    |   movel([0.102355, -1.292766, -2.631086, -0.788537, 1.570796, 1.673152],accel_mss,speed_ms,0,blend_radius_m)
    |   movel([0.101965, -1.293057, -2.630916, -0.788416, 1.570796, 1.672761],accel_mss,speed_ms,0,blend_radius_m)
    |   movel([0.101499, -1.293216, -2.630823, -0.788350, 1.570796, 1.672295],accel_mss,speed_ms,0,blend_radius_m)
    |   movel([0.101150, -1.293383, -2.630725, -0.788281, 1.570796, 1.671947],accel_mss,speed_ms,0,blend_radius_m)
    |   movel([0.100675, -1.293364, -2.630736, -0.788289, 1.570796, 1.671471],accel_mss,speed_ms,0,blend_radius_m)
    |   movel([0.100391, -1.293407, -2.630711, -0.788271, 1.570796, 1.671188],accel_mss,speed_ms,0,blend_radius_m)
    |   movel([0.100053, -1.293699, -2.630540, -0.788150, 1.570796, 1.670849],accel_mss,speed_ms,0,blend_radius_m)
    |   movel([0.100321, -1.293715, -2.630530, -0.788144, 1.570796, 1.671118],accel_mss,speed_ms,0,blend_radius_m)
    |   movel([0.100651, -1.293667, -2.630559, -0.788164, 1.570796, 1.671448],accel_mss,speed_ms,0,blend_radius_m)
    |   movel([0.101031, -1.293650, -2.630569, -0.788171, 1.570796, 1.671827],accel_mss,speed_ms,0,blend_radius_m)
    |   movel([0.101319, -1.293615, -2.630589, -0.788185, 1.570796, 1.672116],accel_mss,speed_ms,0,blend_radius_m)
    |   movel([0.101619, -1.293570, -2.630615, -0.788204, 1.570796, 1.672416],accel_mss,speed_ms,0,blend_radius_m)
    |   movel([0.102043, -1.293494, -2.630660, -0.788235, 1.570796, 1.672840],accel_mss,speed_ms,0,blend_radius_m)
    |   movel([0.101987, -1.293260, -2.630797, -0.788332, 1.570796, 1.672784],accel_mss,speed_ms,0,blend_radius_m)
    |   movel([0.102373, -1.293289, -2.630780, -0.788320, 1.570796, 1.673169],accel_mss,speed_ms,0,blend_radius_m)
    |   movel([0.102475, -1.293491, -2.630662, -0.788236, 1.570796, 1.673271],accel_mss,speed_ms,0,blend_radius_m)
    |   movel([0.102816, -1.293437, -2.630693, -0.788259, 1.570796, 1.673613],accel_mss,speed_ms,0,blend_radius_m)
    |   movel([0.103104, -1.293401, -2.630715, -0.788274, 1.570796, 1.673901],accel_mss,speed_ms,0,blend_radius_m)
    |   movel([0.103382, -1.293344, -2.630748, -0.788297, 1.570796, 1.674178],accel_mss,speed_ms,0,blend_radius_m)
    |   movel([0.103678, -1.293105, -2.630888, -0.788396, 1.570796, 1.674474],accel_mss,speed_ms,0,blend_radius_m)
    |   movel([0.103359, -1.293263, -2.630795, -0.788331, 1.570796, 1.674155],accel_mss,speed_ms,0,blend_radius_m)
    |   movel([0.103194, -1.293136, -2.630870, -0.788383, 1.570796, 1.673991],accel_mss,speed_ms,0,blend_radius_m)
    |   movel([0.103230, -1.292829, -2.631049, -0.788511, 1.570796, 1.674026],accel_mss,speed_ms,0,blend_radius_m)
    |   movel([0.103561, -1.292519, -2.631231, -0.788639, 1.570796, 1.674358],accel_mss,speed_ms,0,blend_radius_m)
    |   movel([0.103869, -1.292455, -2.631268, -0.788666, 1.570796, 1.674665],accel_mss,speed_ms,0,blend_radius_m)
    |   movel([0.103902, -1.292696, -2.631127, -0.788566, 1.570796, 1.674699],accel_mss,speed_ms,0,blend_radius_m)
    |   movel([0.104086, -1.292889, -2.631014, -0.788486, 1.570796, 1.674882],accel_mss,speed_ms,0,blend_radius_m)
    |   movel([0.104470, -1.293089, -2.630897, -0.788403, 1.570796, 1.675266],accel_mss,speed_ms,0,blend_radius_m)
    |   movel([0.104480, -1.293409, -2.630709, -0.788270, 1.570796, 1.675276],accel_mss,speed_ms,0,blend_radius_m)
    |   movel([0.104166, -1.293506, -2.630653, -0.788230, 1.570796, 1.674962],accel_mss,speed_ms,0,blend_radius_m)
    |   movel([0.103943, -1.293445, -2.630688, -0.788255, 1.570796, 1.674739],accel_mss,speed_ms,0,blend_radius_m)
    |   movel([0.103724, -1.293307, -2.630769, -0.788313, 1.570796, 1.674520],accel_mss,speed_ms,0,blend_radius_m)
    |   movel([0.103804, -1.293583, -2.630608, -0.788198, 1.570796, 1.674600],accel_mss,speed_ms,0,blend_radius_m)
    |   movel([0.103792, -1.293977, -2.630377, -0.788035, 1.570796, 1.674589],accel_mss,speed_ms,0,blend_radius_m)
    |   movel([0.103523, -1.294338, -2.630165, -0.787886, 1.570796, 1.674319],accel_mss,speed_ms,0,blend_radius_m)
    |   movel([0.103297, -1.294618, -2.630001, -0.787771, 1.570796, 1.674094],accel_mss,speed_ms,0,blend_radius_m)
    |   movel([0.102982, -1.294687, -2.629960, -0.787742, 1.570796, 1.673778],accel_mss,speed_ms,0,blend_radius_m)
    |   movel([0.102668, -1.294988, -2.629783, -0.787618, 1.570796, 1.673465],accel_mss,speed_ms,0,blend_radius_m)
    |   movel([0.102281, -1.295194, -2.629662, -0.787533, 1.570796, 1.673077],accel_mss,speed_ms,0,blend_radius_m)
    |   movel([0.101902, -1.295350, -2.629570, -0.787469, 1.570796, 1.672698],accel_mss,speed_ms,0,blend_radius_m)
    |   movel([0.101557, -1.295489, -2.629488, -0.787412, 1.570796, 1.672353],accel_mss,speed_ms,0,blend_radius_m)
    |   movel([0.101243, -1.295617, -2.629413, -0.787359, 1.570796, 1.672039],accel_mss,speed_ms,0,blend_radius_m)
    |   movel([0.101286, -1.295842, -2.629280, -0.787267, 1.570796, 1.672083],accel_mss,speed_ms,0,blend_radius_m)
    |   movel([0.100997, -1.295991, -2.629193, -0.787206, 1.570796, 1.671793],accel_mss,speed_ms,0,blend_radius_m)
    |   movel([0.100718, -1.295951, -2.629216, -0.787222, 1.570796, 1.671514],accel_mss,speed_ms,0,blend_radius_m)
    |   movel([0.100425, -1.296077, -2.629142, -0.787170, 1.570796, 1.671222],accel_mss,speed_ms,0,blend_radius_m)
    |   movel([0.099331, -1.296580, -2.628845, -0.786964, 1.570796, 1.670127],accel_mss,speed_ms,0,blend_radius_m)
    |   movel([0.097242, -1.297292, -2.628425, -0.786672, 1.570796, 1.668038],accel_mss,speed_ms,0,blend_radius_m)
    |   movel([0.095038, -1.297963, -2.628028, -0.786398, 1.570796, 1.665834],accel_mss,speed_ms,0,blend_radius_m)
    |   movel([0.093267, -1.298398, -2.627770, -0.786220, 1.570796, 1.664064],accel_mss,speed_ms,0,blend_radius_m)
    |   movel([0.092796, -1.298507, -2.627706, -0.786176, 1.570796, 1.663592],accel_mss,speed_ms,0,blend_radius_m)
    |   movel([0.092505, -1.298577, -2.627664, -0.786148, 1.570796, 1.663301],accel_mss,speed_ms,0,blend_radius_m)
    |   movel([0.092006, -1.298695, -2.627594, -0.786099, 1.570796, 1.662802],accel_mss,speed_ms,0,blend_radius_m)
    |   movel([0.091686, -1.298709, -2.627586, -0.786094, 1.570796, 1.662483],accel_mss,speed_ms,0,blend_radius_m)
    |   movel([0.091516, -1.298549, -2.627681, -0.786159, 1.570796, 1.662312],accel_mss,speed_ms,0,blend_radius_m)
    |   movel([0.090908, -1.298604, -2.627648, -0.786137, 1.570796, 1.661704],accel_mss,speed_ms,0,blend_radius_m)
    |   movel([0.091012, -1.298791, -2.627537, -0.786060, 1.570796, 1.661808],accel_mss,speed_ms,0,blend_radius_m)
    |   movel([0.091131, -1.298957, -2.627439, -0.785993, 1.570796, 1.661927],accel_mss,speed_ms,0,blend_radius_m)
    |   movel([0.091380, -1.299030, -2.627396, -0.785963, 1.570796, 1.662176],accel_mss,speed_ms,0,blend_radius_m)
    |   movel([0.091703, -1.299034, -2.627394, -0.785962, 1.570796, 1.662500],accel_mss,speed_ms,0,blend_radius_m)
    |   movel([0.091970, -1.298785, -2.627541, -0.786063, 1.570796, 1.662766],accel_mss,speed_ms,0,blend_radius_m)
    |   movel([0.092331, -1.298807, -2.627528, -0.786054, 1.570796, 1.663127],accel_mss,speed_ms,0,blend_radius_m)
    |   movel([0.092659, -1.298717, -2.627581, -0.786090, 1.570796, 1.663455],accel_mss,speed_ms,0,blend_radius_m)
    |   movel([0.092762, -1.298900, -2.627473, -0.786016, 1.570796, 1.663559],accel_mss,speed_ms,0,blend_radius_m)
    |   movel([0.092991, -1.298961, -2.627436, -0.785991, 1.570796, 1.663787],accel_mss,speed_ms,0,blend_radius_m)
    |   movel([0.093296, -1.298783, -2.627542, -0.786064, 1.570796, 1.664092],accel_mss,speed_ms,0,blend_radius_m)
    |   movel([0.093554, -1.298769, -2.627551, -0.786070, 1.570796, 1.664350],accel_mss,speed_ms,0,blend_radius_m)
    |   movel([0.093259, -1.299029, -2.627397, -0.785964, 1.570796, 1.664056],accel_mss,speed_ms,0,blend_radius_m)
    |   movel([0.092956, -1.299112, -2.627347, -0.785930, 1.570796, 1.663753],accel_mss,speed_ms,0,blend_radius_m)
    |   movel([0.092691, -1.299070, -2.627372, -0.785947, 1.570796, 1.663487],accel_mss,speed_ms,0,blend_radius_m)
    |   movel([0.092356, -1.298978, -2.627427, -0.785984, 1.570796, 1.663152],accel_mss,speed_ms,0,blend_radius_m)
    |   movel([0.092063, -1.299023, -2.627400, -0.785966, 1.570796, 1.662859],accel_mss,speed_ms,0,blend_radius_m)
    |   movel([0.091652, -1.299143, -2.627329, -0.785917, 1.570796, 1.662448],accel_mss,speed_ms,0,blend_radius_m)
    |   movel([0.091327, -1.299231, -2.627276, -0.785881, 1.570796, 1.662123],accel_mss,speed_ms,0,blend_radius_m)
    |   movel([0.091035, -1.299288, -2.627243, -0.785858, 1.570796, 1.661832],accel_mss,speed_ms,0,blend_radius_m)
    |   movel([0.090721, -1.299331, -2.627217, -0.785841, 1.570796, 1.661517],accel_mss,speed_ms,0,blend_radius_m)
    |   movel([0.090684, -1.299094, -2.627358, -0.785937, 1.570796, 1.661480],accel_mss,speed_ms,0,blend_radius_m)
    |   movel([0.090510, -1.298965, -2.627434, -0.785990, 1.570796, 1.661306],accel_mss,speed_ms,0,blend_radius_m)
    |   movel([0.090188, -1.299079, -2.627367, -0.785943, 1.570796, 1.660984],accel_mss,speed_ms,0,blend_radius_m)
    |   movel([0.090012, -1.298940, -2.627449, -0.786000, 1.570796, 1.660808],accel_mss,speed_ms,0,blend_radius_m)
    |   movel([0.089943, -1.298729, -2.627574, -0.786086, 1.570796, 1.660739],accel_mss,speed_ms,0,blend_radius_m)
    |   movel([0.089712, -1.298679, -2.627604, -0.786106, 1.570796, 1.660509],accel_mss,speed_ms,0,blend_radius_m)
    |   movel([0.089970, -1.298437, -2.627747, -0.786205, 1.570796, 1.660766],accel_mss,speed_ms,0,blend_radius_m)
    |   movel([0.090285, -1.298394, -2.627773, -0.786222, 1.570796, 1.661081],accel_mss,speed_ms,0,blend_radius_m)
    |   movel([0.090132, -1.298683, -2.627602, -0.786105, 1.570796, 1.660928],accel_mss,speed_ms,0,blend_radius_m)
    |   movel([0.090205, -1.298963, -2.627436, -0.785991, 1.570796, 1.661001],accel_mss,speed_ms,0,blend_radius_m)
    |   movel([0.090261, -1.298678, -2.627605, -0.786107, 1.570796, 1.661057],accel_mss,speed_ms,0,blend_radius_m)
    |   movel([0.090563, -1.298554, -2.627678, -0.786157, 1.570796, 1.661359],accel_mss,speed_ms,0,blend_radius_m)
    |   movel([0.090470, -1.298342, -2.627804, -0.786244, 1.570796, 1.661266],accel_mss,speed_ms,0,blend_radius_m)
    |   movel([0.090383, -1.298068, -2.627966, -0.786355, 1.570796, 1.661179],accel_mss,speed_ms,0,blend_radius_m)
    |   movel([0.090678, -1.297826, -2.628109, -0.786454, 1.570796, 1.661474],accel_mss,speed_ms,0,blend_radius_m)
    |   movel([0.090825, -1.297494, -2.628306, -0.786590, 1.570796, 1.661621],accel_mss,speed_ms,0,blend_radius_m)
    |   movel([0.090518, -1.297690, -2.628189, -0.786509, 1.570796, 1.661314],accel_mss,speed_ms,0,blend_radius_m)
    |   movel([0.090290, -1.297927, -2.628049, -0.786413, 1.570796, 1.661086],accel_mss,speed_ms,0,blend_radius_m)
    |   movel([0.090113, -1.298212, -2.627880, -0.786296, 1.570796, 1.660910],accel_mss,speed_ms,0,blend_radius_m)
    |   movel([0.089804, -1.298280, -2.627840, -0.786269, 1.570796, 1.660600],accel_mss,speed_ms,0,blend_radius_m)
    |   movel([0.089954, -1.297963, -2.628028, -0.786398, 1.570796, 1.660750],accel_mss,speed_ms,0,blend_radius_m)
    |   movel([0.090167, -1.297691, -2.628189, -0.786509, 1.570796, 1.660963],accel_mss,speed_ms,0,blend_radius_m)
    |   movel([0.090457, -1.297347, -2.628392, -0.786650, 1.570796, 1.661253],accel_mss,speed_ms,0,blend_radius_m)
    |   movel([0.090350, -1.297056, -2.628564, -0.786769, 1.570796, 1.661146],accel_mss,speed_ms,0,blend_radius_m)
    |   movel([0.090002, -1.296971, -2.628614, -0.786803, 1.570796, 1.660798],accel_mss,speed_ms,0,blend_radius_m)
    |   movel([0.089628, -1.296935, -2.628635, -0.786818, 1.570796, 1.660424],accel_mss,speed_ms,0,blend_radius_m)
    |   movel([0.089304, -1.296977, -2.628611, -0.786801, 1.570796, 1.660101],accel_mss,speed_ms,0,blend_radius_m)
    |   movel([0.089032, -1.296934, -2.628637, -0.786819, 1.570796, 1.659829],accel_mss,speed_ms,0,blend_radius_m)
    |   movel([0.088749, -1.296974, -2.628613, -0.786802, 1.570796, 1.659546],accel_mss,speed_ms,0,blend_radius_m)
    |   movel([0.088519, -1.296916, -2.628647, -0.786826, 1.570796, 1.659315],accel_mss,speed_ms,0,blend_radius_m)
    |   movel([0.088260, -1.296793, -2.628720, -0.786877, 1.570796, 1.659057],accel_mss,speed_ms,0,blend_radius_m)
    |   movel([0.087984, -1.296604, -2.628831, -0.786954, 1.570796, 1.658780],accel_mss,speed_ms,0,blend_radius_m)
    |   movel([0.087838, -1.296402, -2.628950, -0.787037, 1.570796, 1.658634],accel_mss,speed_ms,0,blend_radius_m)
    |   movel([0.087930, -1.296130, -2.629111, -0.787148, 1.570796, 1.658726],accel_mss,speed_ms,0,blend_radius_m)
    |   movel([0.088018, -1.295835, -2.629284, -0.787270, 1.570796, 1.658814],accel_mss,speed_ms,0,blend_radius_m)
    |   movel([0.088177, -1.295298, -2.629600, -0.787490, 1.570796, 1.658973],accel_mss,speed_ms,0,blend_radius_m)
    |   movel([0.088520, -1.294882, -2.629845, -0.787662, 1.570796, 1.659316],accel_mss,speed_ms,0,blend_radius_m)
    |   movel([0.088850, -1.294590, -2.630017, -0.787782, 1.570796, 1.659647],accel_mss,speed_ms,0,blend_radius_m)
    |   movel([0.089096, -1.294365, -2.630149, -0.787875, 1.570796, 1.659893],accel_mss,speed_ms,0,blend_radius_m)
    |   movel([0.089150, -1.293993, -2.630367, -0.788029, 1.570796, 1.659946],accel_mss,speed_ms,0,blend_radius_m)
    |   movel([0.088850, -1.293957, -2.630389, -0.788044, 1.570796, 1.659646],accel_mss,speed_ms,0,blend_radius_m)
    |   movel([0.088651, -1.293819, -2.630469, -0.788100, 1.570796, 1.659447],accel_mss,speed_ms,0,blend_radius_m)
    |   movel([0.088309, -1.293899, -2.630422, -0.788068, 1.570796, 1.659105],accel_mss,speed_ms,0,blend_radius_m)
    |   movel([0.087687, -1.293983, -2.630373, -0.788033, 1.570796, 1.658483],accel_mss,speed_ms,0,blend_radius_m)
    |   movel([0.087026, -1.293852, -2.630450, -0.788087, 1.570796, 1.657823],accel_mss,speed_ms,0,blend_radius_m)
    |   movel([0.086481, -1.293564, -2.630619, -0.788206, 1.570796, 1.657277],accel_mss,speed_ms,0,blend_radius_m)
    |   movel([0.086205, -1.293166, -2.630852, -0.788371, 1.570796, 1.657001],accel_mss,speed_ms,0,blend_radius_m)
    |   movel([0.086167, -1.292865, -2.631028, -0.788496, 1.570796, 1.656963],accel_mss,speed_ms,0,blend_radius_m)
    |   movel([0.086235, -1.292549, -2.631213, -0.788627, 1.570796, 1.657032],accel_mss,speed_ms,0,blend_radius_m)
    |   movel([0.086426, -1.292178, -2.631430, -0.788781, 1.570796, 1.657222],accel_mss,speed_ms,0,blend_radius_m)
    |   movel([0.086757, -1.291717, -2.631699, -0.788973, 1.570796, 1.657553],accel_mss,speed_ms,0,blend_radius_m)
    |   movel([0.086981, -1.291477, -2.631839, -0.789073, 1.570796, 1.657777],accel_mss,speed_ms,0,blend_radius_m)
    |   movel([0.087305, -1.291207, -2.631997, -0.789185, 1.570796, 1.658101],accel_mss,speed_ms,0,blend_radius_m)
    |   movel([0.087627, -1.290981, -2.632129, -0.789279, 1.570796, 1.658423],accel_mss,speed_ms,0,blend_radius_m)
    |   movel([0.087930, -1.290792, -2.632238, -0.789358, 1.570796, 1.658726],accel_mss,speed_ms,0,blend_radius_m)
    |   movel([0.088216, -1.290788, -2.632241, -0.789360, 1.570796, 1.659013],accel_mss,speed_ms,0,blend_radius_m)
    |   movel([0.088406, -1.290922, -2.632163, -0.789304, 1.570796, 1.659202],accel_mss,speed_ms,0,blend_radius_m)
    |   movel([0.088248, -1.290579, -2.632363, -0.789447, 1.570796, 1.659044],accel_mss,speed_ms,0,blend_radius_m)
    |   movel([0.088513, -1.290389, -2.632473, -0.789526, 1.570796, 1.659309],accel_mss,speed_ms,0,blend_radius_m)
    |   movel([0.088853, -1.290071, -2.632658, -0.789660, 1.570796, 1.659650],accel_mss,speed_ms,0,blend_radius_m)
    |   movel([0.089467, -1.289643, -2.632907, -0.789839, 1.570796, 1.660263],accel_mss,speed_ms,0,blend_radius_m)
    |   movel([0.090092, -1.289248, -2.633137, -0.790004, 1.570796, 1.660888],accel_mss,speed_ms,0,blend_radius_m)
    |   movel([0.090426, -1.289175, -2.633179, -0.790035, 1.570796, 1.661223],accel_mss,speed_ms,0,blend_radius_m)
    |   movel([0.090517, -1.289419, -2.633037, -0.789932, 1.570796, 1.661314],accel_mss,speed_ms,0,blend_radius_m)
    |   speed_ms = 0.003
    |   movel([0.090517, -1.275491, -2.626410, -0.810488, 1.570796, 1.661314],accel_mss,speed_ms,0,blend_radius_m)
    |   speed_ms = 1.000
    |   movel([0.090517, -1.248993, -2.612771, -0.850625, 1.570796, 1.661314],accel_mss,speed_ms,0,blend_radius_m)
    |   movel([0.108394, -1.243984, -2.615506, -0.852900, 1.570796, 1.679191],accel_mss,speed_ms,0,blend_radius_m)
    |   movel([0.108394, -1.270545, -2.629211, -0.812633, 1.570796, 1.679191],accel_mss,speed_ms,0,blend_radius_m)
    |   speed_ms = 0.003
    |   movel([0.108394, -1.280978, -2.634218, -0.797193, 1.570796, 1.679191],accel_mss,speed_ms,0,blend_radius_m)
    |   speed_ms = 0.007
    |   movel([0.108672, -1.280919, -2.634252, -0.797218, 1.570796, 1.679468],accel_mss,speed_ms,0,blend_radius_m)
    |   movel([0.108972, -1.280870, -2.634280, -0.797239, 1.570796, 1.679768],accel_mss,speed_ms,0,blend_radius_m)
    |   movel([0.108590, -1.281076, -2.634162, -0.797151, 1.570796, 1.679387],accel_mss,speed_ms,0,blend_radius_m)
    |   movel([0.108394, -1.280978, -2.634218, -0.797193, 1.570796, 1.679191],accel_mss,speed_ms,0,blend_radius_m)
    |   speed_ms = 0.003
    |   movel([0.108394, -1.284514, -2.635871, -0.792004, 1.570796, 1.679191],accel_mss,speed_ms,0,blend_radius_m)
    |   speed_ms = 0.007
    |   movel([0.108672, -1.284455, -2.635905, -0.792029, 1.570796, 1.679468],accel_mss,speed_ms,0,blend_radius_m)
    |   movel([0.108972, -1.284406, -2.635933, -0.792050, 1.570796, 1.679768],accel_mss,speed_ms,0,blend_radius_m)
    |   movel([0.108590, -1.284612, -2.635815, -0.791962, 1.570796, 1.679387],accel_mss,speed_ms,0,blend_radius_m)
    |   movel([0.108394, -1.284514, -2.635871, -0.792004, 1.570796, 1.679191],accel_mss,speed_ms,0,blend_radius_m)
    |   speed_ms = 0.003
    |   movel([0.108394, -1.270545, -2.629211, -0.812633, 1.570796, 1.679191],accel_mss,speed_ms,0,blend_radius_m)
    |   speed_ms = 1.000
    |   movel([0.108394, -1.243984, -2.615506, -0.852900, 1.570796, 1.679191],accel_mss,speed_ms,0,blend_radius_m)
    |   movel([0.134199, -1.228063, -2.624004, -0.860322, 1.570796, 1.704996],accel_mss,speed_ms,0,blend_radius_m)
    |   movel([0.134199, -1.254817, -2.637919, -0.819653, 1.570796, 1.704996],accel_mss,speed_ms,0,blend_radius_m)
    |   speed_ms = 0.003
    |   movel([0.134199, -1.265339, -2.643007, -0.804044, 1.570796, 1.704996],accel_mss,speed_ms,0,blend_radius_m)
    |   speed_ms = 0.007
    |   movel([0.134398, -1.265029, -2.643178, -0.804183, 1.570796, 1.705194],accel_mss,speed_ms,0,blend_radius_m)
    |   movel([0.134745, -1.264784, -2.643313, -0.804292, 1.570796, 1.705541],accel_mss,speed_ms,0,blend_radius_m)
    |   movel([0.135237, -1.264642, -2.643391, -0.804356, 1.570796, 1.706033],accel_mss,speed_ms,0,blend_radius_m)
    |   movel([0.135651, -1.264639, -2.643393, -0.804357, 1.570796, 1.706448],accel_mss,speed_ms,0,blend_radius_m)
    |   movel([0.135748, -1.264848, -2.643278, -0.804264, 1.570796, 1.706545],accel_mss,speed_ms,0,blend_radius_m)
    |   movel([0.135483, -1.265183, -2.643092, -0.804113, 1.570796, 1.706279],accel_mss,speed_ms,0,blend_radius_m)
    |   movel([0.135213, -1.265424, -2.642960, -0.804005, 1.570796, 1.706009],accel_mss,speed_ms,0,blend_radius_m)
    |   movel([0.134898, -1.265584, -2.642871, -0.803934, 1.570796, 1.705694],accel_mss,speed_ms,0,blend_radius_m)
    |   movel([0.134599, -1.265633, -2.642844, -0.803912, 1.570796, 1.705396],accel_mss,speed_ms,0,blend_radius_m)
    |   movel([0.134371, -1.265561, -2.642884, -0.803944, 1.570796, 1.705167],accel_mss,speed_ms,0,blend_radius_m)
    |   movel([0.134199, -1.265339, -2.643007, -0.804044, 1.570796, 1.704996],accel_mss,speed_ms,0,blend_radius_m)
    |   speed_ms = 0.003
    |   movel([0.134199, -1.268907, -2.644686, -0.798796, 1.570796, 1.704996],accel_mss,speed_ms,0,blend_radius_m)
    |   speed_ms = 0.007
    |   movel([0.134398, -1.268597, -2.644858, -0.798934, 1.570796, 1.705194],accel_mss,speed_ms,0,blend_radius_m)
    |   movel([0.134745, -1.268352, -2.644993, -0.799043, 1.570796, 1.705541],accel_mss,speed_ms,0,blend_radius_m)
    |   movel([0.135237, -1.268211, -2.645072, -0.799106, 1.570796, 1.706033],accel_mss,speed_ms,0,blend_radius_m)
    |   movel([0.135651, -1.268209, -2.645073, -0.799107, 1.570796, 1.706448],accel_mss,speed_ms,0,blend_radius_m)
    |   movel([0.135748, -1.268416, -2.644958, -0.799015, 1.570796, 1.706545],accel_mss,speed_ms,0,blend_radius_m)
    |   movel([0.135483, -1.268752, -2.644772, -0.798865, 1.570796, 1.706279],accel_mss,speed_ms,0,blend_radius_m)
    |   movel([0.135213, -1.268992, -2.644639, -0.798758, 1.570796, 1.706009],accel_mss,speed_ms,0,blend_radius_m)
    |   movel([0.134898, -1.269152, -2.644550, -0.798687, 1.570796, 1.705694],accel_mss,speed_ms,0,blend_radius_m)
    |   movel([0.134599, -1.269200, -2.644523, -0.798666, 1.570796, 1.705396],accel_mss,speed_ms,0,blend_radius_m)
    |   movel([0.134371, -1.269128, -2.644563, -0.798698, 1.570796, 1.705167],accel_mss,speed_ms,0,blend_radius_m)
    |   movel([0.134199, -1.268907, -2.644686, -0.798796, 1.570796, 1.704996],accel_mss,speed_ms,0,blend_radius_m)
    |   speed_ms = 0.003
    |   movel([0.134199, -1.254817, -2.637919, -0.819653, 1.570796, 1.704996],accel_mss,speed_ms,0,blend_radius_m)
    |   speed_ms = 1.000
    |   movel([0.134199, -1.228063, -2.624004, -0.860322, 1.570796, 1.704996],accel_mss,speed_ms,0,blend_radius_m)
    |   movel([0.135018, -1.226764, -2.624685, -0.860940, 1.570796, 1.705815],accel_mss,speed_ms,0,blend_radius_m)
    |   movel([0.135018, -1.253533, -2.638617, -0.820240, 1.570796, 1.705815],accel_mss,speed_ms,0,blend_radius_m)
    |   speed_ms = 0.003
    |   movel([0.135018, -1.264062, -2.643711, -0.804616, 1.570796, 1.705815],accel_mss,speed_ms,0,blend_radius_m)
    |   speed_ms = 0.007
    |   movel([0.133569, -1.264514, -2.643462, -0.804413, 1.570796, 1.704366],accel_mss,speed_ms,0,blend_radius_m)
    |   movel([0.132754, -1.264606, -2.643411, -0.804372, 1.570796, 1.703551],accel_mss,speed_ms,0,blend_radius_m)
    |   movel([0.132393, -1.264541, -2.643447, -0.804401, 1.570796, 1.703189],accel_mss,speed_ms,0,blend_radius_m)
    |   movel([0.132220, -1.264399, -2.643525, -0.804465, 1.570796, 1.703016],accel_mss,speed_ms,0,blend_radius_m)
    |   movel([0.132406, -1.263908, -2.643795, -0.804685, 1.570796, 1.703203],accel_mss,speed_ms,0,blend_radius_m)
    |   movel([0.132616, -1.263631, -2.643948, -0.804810, 1.570796, 1.703412],accel_mss,speed_ms,0,blend_radius_m)
    |   movel([0.132602, -1.263320, -2.644119, -0.804950, 1.570796, 1.703398],accel_mss,speed_ms,0,blend_radius_m)
    |   movel([0.132363, -1.263216, -2.644176, -0.804997, 1.570796, 1.703159],accel_mss,speed_ms,0,blend_radius_m)
    |   movel([0.132010, -1.263108, -2.644235, -0.805045, 1.570796, 1.702806],accel_mss,speed_ms,0,blend_radius_m)
    |   movel([0.132437, -1.262707, -2.644456, -0.805226, 1.570796, 1.703234],accel_mss,speed_ms,0,blend_radius_m)
    |   movel([0.132758, -1.262384, -2.644633, -0.805372, 1.570796, 1.703554],accel_mss,speed_ms,0,blend_radius_m)
    |   movel([0.132813, -1.262065, -2.644808, -0.805516, 1.570796, 1.703609],accel_mss,speed_ms,0,blend_radius_m)
    |   movel([0.132580, -1.261897, -2.644900, -0.805592, 1.570796, 1.703377],accel_mss,speed_ms,0,blend_radius_m)
    |   movel([0.132378, -1.261707, -2.645004, -0.805678, 1.570796, 1.703175],accel_mss,speed_ms,0,blend_radius_m)
    |   movel([0.132314, -1.261470, -2.645134, -0.805785, 1.570796, 1.703111],accel_mss,speed_ms,0,blend_radius_m)
    |   movel([0.132399, -1.261194, -2.645285, -0.805910, 1.570796, 1.703195],accel_mss,speed_ms,0,blend_radius_m)
    |   movel([0.132615, -1.260893, -2.645450, -0.806046, 1.570796, 1.703411],accel_mss,speed_ms,0,blend_radius_m)
    |   movel([0.132980, -1.260625, -2.645596, -0.806168, 1.570796, 1.703776],accel_mss,speed_ms,0,blend_radius_m)
    |   movel([0.133606, -1.260445, -2.645695, -0.806250, 1.570796, 1.704403],accel_mss,speed_ms,0,blend_radius_m)
    |   movel([0.134003, -1.260357, -2.645743, -0.806289, 1.570796, 1.704799],accel_mss,speed_ms,0,blend_radius_m)
    |   movel([0.134688, -1.260200, -2.645828, -0.806361, 1.570796, 1.705485],accel_mss,speed_ms,0,blend_radius_m)
    |   movel([0.135480, -1.260013, -2.645930, -0.806446, 1.570796, 1.706276],accel_mss,speed_ms,0,blend_radius_m)
    |   movel([0.136283, -1.259823, -2.646034, -0.806532, 1.570796, 1.707080],accel_mss,speed_ms,0,blend_radius_m)
    |   movel([0.137293, -1.259591, -2.646161, -0.806637, 1.570796, 1.708089],accel_mss,speed_ms,0,blend_radius_m)
    |   movel([0.137906, -1.259479, -2.646222, -0.806688, 1.570796, 1.708703],accel_mss,speed_ms,0,blend_radius_m)
    |   movel([0.138308, -1.259446, -2.646240, -0.806703, 1.570796, 1.709104],accel_mss,speed_ms,0,blend_radius_m)
    |   movel([0.138558, -1.259495, -2.646213, -0.806681, 1.570796, 1.709354],accel_mss,speed_ms,0,blend_radius_m)
    |   movel([0.138772, -1.259631, -2.646139, -0.806619, 1.570796, 1.709569],accel_mss,speed_ms,0,blend_radius_m)
    |   movel([0.138742, -1.260008, -2.645933, -0.806448, 1.570796, 1.709538],accel_mss,speed_ms,0,blend_radius_m)
    |   movel([0.138459, -1.260449, -2.645692, -0.806248, 1.570796, 1.709255],accel_mss,speed_ms,0,blend_radius_m)
    |   movel([0.138261, -1.260761, -2.645522, -0.806106, 1.570796, 1.709057],accel_mss,speed_ms,0,blend_radius_m)
    |   movel([0.138159, -1.261142, -2.645313, -0.805933, 1.570796, 1.708956],accel_mss,speed_ms,0,blend_radius_m)
    |   movel([0.138212, -1.261391, -2.645178, -0.805821, 1.570796, 1.709008],accel_mss,speed_ms,0,blend_radius_m)
    |   movel([0.138231, -1.261781, -2.644964, -0.805644, 1.570796, 1.709028],accel_mss,speed_ms,0,blend_radius_m)
    |   movel([0.138086, -1.262178, -2.644746, -0.805465, 1.570796, 1.708883],accel_mss,speed_ms,0,blend_radius_m)
    |   movel([0.137764, -1.262595, -2.644517, -0.805277, 1.570796, 1.708560],accel_mss,speed_ms,0,blend_radius_m)
    |   movel([0.137253, -1.263048, -2.644269, -0.805072, 1.570796, 1.708050],accel_mss,speed_ms,0,blend_radius_m)
    |   movel([0.136472, -1.263511, -2.644014, -0.804864, 1.570796, 1.707268],accel_mss,speed_ms,0,blend_radius_m)
    |   movel([0.135018, -1.264062, -2.643711, -0.804616, 1.570796, 1.705815],accel_mss,speed_ms,0,blend_radius_m)
    |   speed_ms = 0.003
    |   movel([0.135018, -1.267632, -2.645392, -0.799364, 1.570796, 1.705815],accel_mss,speed_ms,0,blend_radius_m)
    |   speed_ms = 0.007
    |   movel([0.133569, -1.268083, -2.645143, -0.799163, 1.570796, 1.704366],accel_mss,speed_ms,0,blend_radius_m)
    |   movel([0.132754, -1.268175, -2.645092, -0.799122, 1.570796, 1.703551],accel_mss,speed_ms,0,blend_radius_m)
    |   movel([0.132393, -1.268110, -2.645128, -0.799151, 1.570796, 1.703189],accel_mss,speed_ms,0,blend_radius_m)
    |   movel([0.132220, -1.267969, -2.645206, -0.799214, 1.570796, 1.703016],accel_mss,speed_ms,0,blend_radius_m)
    |   movel([0.132406, -1.267479, -2.645477, -0.799433, 1.570796, 1.703203],accel_mss,speed_ms,0,blend_radius_m)
    |   movel([0.132616, -1.267202, -2.645630, -0.799557, 1.570796, 1.703412],accel_mss,speed_ms,0,blend_radius_m)
    |   movel([0.132602, -1.266891, -2.645802, -0.799695, 1.570796, 1.703398],accel_mss,speed_ms,0,blend_radius_m)
    |   movel([0.132363, -1.266788, -2.645859, -0.799742, 1.570796, 1.703159],accel_mss,speed_ms,0,blend_radius_m)
    |   movel([0.132010, -1.266681, -2.645919, -0.799790, 1.570796, 1.702806],accel_mss,speed_ms,0,blend_radius_m)
    |   movel([0.132437, -1.266280, -2.646140, -0.799969, 1.570796, 1.703234],accel_mss,speed_ms,0,blend_radius_m)
    |   movel([0.132758, -1.265958, -2.646318, -0.800114, 1.570796, 1.703554],accel_mss,speed_ms,0,blend_radius_m)
    |   movel([0.132813, -1.265640, -2.646493, -0.800256, 1.570796, 1.703609],accel_mss,speed_ms,0,blend_radius_m)
    |   movel([0.132580, -1.265472, -2.646585, -0.800332, 1.570796, 1.703377],accel_mss,speed_ms,0,blend_radius_m)
    |   movel([0.132378, -1.265282, -2.646690, -0.800417, 1.570796, 1.703175],accel_mss,speed_ms,0,blend_radius_m)
    |   movel([0.132314, -1.265045, -2.646820, -0.800523, 1.570796, 1.703111],accel_mss,speed_ms,0,blend_radius_m)
    |   movel([0.132399, -1.264770, -2.646972, -0.800647, 1.570796, 1.703195],accel_mss,speed_ms,0,blend_radius_m)
    |   movel([0.132615, -1.264470, -2.647137, -0.800782, 1.570796, 1.703411],accel_mss,speed_ms,0,blend_radius_m)
    |   movel([0.132980, -1.264202, -2.647284, -0.800903, 1.570796, 1.703776],accel_mss,speed_ms,0,blend_radius_m)
    |   movel([0.133606, -1.264022, -2.647383, -0.800984, 1.570796, 1.704403],accel_mss,speed_ms,0,blend_radius_m)
    |   movel([0.134003, -1.263934, -2.647431, -0.801024, 1.570796, 1.704799],accel_mss,speed_ms,0,blend_radius_m)
    |   movel([0.134688, -1.263778, -2.647517, -0.801094, 1.570796, 1.705485],accel_mss,speed_ms,0,blend_radius_m)
    |   movel([0.135480, -1.263591, -2.647619, -0.801179, 1.570796, 1.706276],accel_mss,speed_ms,0,blend_radius_m)
    |   movel([0.136283, -1.263401, -2.647723, -0.801264, 1.570796, 1.707080],accel_mss,speed_ms,0,blend_radius_m)
    |   movel([0.137293, -1.263170, -2.647850, -0.801369, 1.570796, 1.708089],accel_mss,speed_ms,0,blend_radius_m)
    |   movel([0.137906, -1.263058, -2.647911, -0.801420, 1.570796, 1.708703],accel_mss,speed_ms,0,blend_radius_m)
    |   movel([0.138308, -1.263025, -2.647930, -0.801435, 1.570796, 1.709104],accel_mss,speed_ms,0,blend_radius_m)
    |   movel([0.138558, -1.263074, -2.647902, -0.801412, 1.570796, 1.709354],accel_mss,speed_ms,0,blend_radius_m)
    |   movel([0.138772, -1.263210, -2.647828, -0.801351, 1.570796, 1.709569],accel_mss,speed_ms,0,blend_radius_m)
    |   movel([0.138742, -1.263586, -2.647622, -0.801181, 1.570796, 1.709538],accel_mss,speed_ms,0,blend_radius_m)
    |   movel([0.138459, -1.264027, -2.647380, -0.800982, 1.570796, 1.709255],accel_mss,speed_ms,0,blend_radius_m)
    |   movel([0.138261, -1.264338, -2.647209, -0.800842, 1.570796, 1.709057],accel_mss,speed_ms,0,blend_radius_m)
    |   movel([0.138159, -1.264718, -2.647000, -0.800671, 1.570796, 1.708956],accel_mss,speed_ms,0,blend_radius_m)
    |   movel([0.138212, -1.264966, -2.646864, -0.800559, 1.570796, 1.709008],accel_mss,speed_ms,0,blend_radius_m)
    |   movel([0.138231, -1.265356, -2.646649, -0.800384, 1.570796, 1.709028],accel_mss,speed_ms,0,blend_radius_m)
    |   movel([0.138086, -1.265752, -2.646431, -0.800206, 1.570796, 1.708883],accel_mss,speed_ms,0,blend_radius_m)
    |   movel([0.137764, -1.266168, -2.646201, -0.800019, 1.570796, 1.708560],accel_mss,speed_ms,0,blend_radius_m)
    |   movel([0.137253, -1.266620, -2.645952, -0.799817, 1.570796, 1.708050],accel_mss,speed_ms,0,blend_radius_m)
    |   movel([0.136472, -1.267082, -2.645697, -0.799610, 1.570796, 1.707268],accel_mss,speed_ms,0,blend_radius_m)
    |   movel([0.135018, -1.267632, -2.645392, -0.799364, 1.570796, 1.705815],accel_mss,speed_ms,0,blend_radius_m)
    |   speed_ms = 0.003
    |   movel([0.135018, -1.253533, -2.638617, -0.820240, 1.570796, 1.705815],accel_mss,speed_ms,0,blend_radius_m)
    |   speed_ms = 1.000
    |   movel([0.135018, -1.226764, -2.624685, -0.860940, 1.570796, 1.705815],accel_mss,speed_ms,0,blend_radius_m)
    |   movel([0.137358, -1.221519, -2.627413, -0.863457, 1.570796, 1.708154],accel_mss,speed_ms,0,blend_radius_m)
    |   movel([0.137358, -1.248347, -2.641414, -0.822628, 1.570796, 1.708154],accel_mss,speed_ms,0,blend_radius_m)
    |   speed_ms = 0.003
    |   movel([0.137358, -1.258904, -2.646535, -0.806950, 1.570796, 1.708154],accel_mss,speed_ms,0,blend_radius_m)
    |   speed_ms = 0.007
    |   movel([0.137144, -1.258616, -2.646692, -0.807081, 1.570796, 1.707940],accel_mss,speed_ms,0,blend_radius_m)
    |   movel([0.137235, -1.257961, -2.647048, -0.807380, 1.570796, 1.708031],accel_mss,speed_ms,0,blend_radius_m)
    |   movel([0.137436, -1.256880, -2.647634, -0.807874, 1.570796, 1.708233],accel_mss,speed_ms,0,blend_radius_m)
    |   movel([0.137871, -1.254806, -2.648756, -0.808827, 1.570796, 1.708667],accel_mss,speed_ms,0,blend_radius_m)
    |   movel([0.138200, -1.253306, -2.649563, -0.809519, 1.570796, 1.708997],accel_mss,speed_ms,0,blend_radius_m)
    |   movel([0.138501, -1.252015, -2.650256, -0.810117, 1.570796, 1.709297],accel_mss,speed_ms,0,blend_radius_m)
    |   movel([0.138778, -1.250887, -2.650861, -0.810642, 1.570796, 1.709574],accel_mss,speed_ms,0,blend_radius_m)
    |   movel([0.139175, -1.250471, -2.651083, -0.810835, 1.570796, 1.709971],accel_mss,speed_ms,0,blend_radius_m)
    |   movel([0.139446, -1.250254, -2.651199, -0.810936, 1.570796, 1.710242],accel_mss,speed_ms,0,blend_radius_m)
    |   movel([0.139737, -1.250029, -2.651319, -0.811041, 1.570796, 1.710534],accel_mss,speed_ms,0,blend_radius_m)
    |   movel([0.140340, -1.249523, -2.651589, -0.811277, 1.570796, 1.711136],accel_mss,speed_ms,0,blend_radius_m)
    |   movel([0.140778, -1.249049, -2.651841, -0.811499, 1.570796, 1.711574],accel_mss,speed_ms,0,blend_radius_m)
    |   movel([0.141088, -1.248562, -2.652101, -0.811727, 1.570796, 1.711885],accel_mss,speed_ms,0,blend_radius_m)
    |   movel([0.141299, -1.248024, -2.652387, -0.811978, 1.570796, 1.712095],accel_mss,speed_ms,0,blend_radius_m)
    |   movel([0.141376, -1.247686, -2.652566, -0.812137, 1.570796, 1.712172],accel_mss,speed_ms,0,blend_radius_m)
    |   movel([0.141270, -1.247330, -2.652755, -0.812304, 1.570796, 1.712067],accel_mss,speed_ms,0,blend_radius_m)
    |   movel([0.141024, -1.247133, -2.652860, -0.812396, 1.570796, 1.711820],accel_mss,speed_ms,0,blend_radius_m)
    |   movel([0.140322, -1.246938, -2.652963, -0.812488, 1.570796, 1.711118],accel_mss,speed_ms,0,blend_radius_m)
    |   movel([0.139577, -1.247221, -2.652813, -0.812355, 1.570796, 1.710374],accel_mss,speed_ms,0,blend_radius_m)
    |   movel([0.138926, -1.247946, -2.652428, -0.812015, 1.570796, 1.709723],accel_mss,speed_ms,0,blend_radius_m)
    |   movel([0.138497, -1.248983, -2.651876, -0.811529, 1.570796, 1.709294],accel_mss,speed_ms,0,blend_radius_m)
    |   movel([0.138299, -1.249669, -2.651511, -0.811209, 1.570796, 1.709096],accel_mss,speed_ms,0,blend_radius_m)
    |   movel([0.138115, -1.250027, -2.651320, -0.811042, 1.570796, 1.708911],accel_mss,speed_ms,0,blend_radius_m)
    |   movel([0.137451, -1.250470, -2.651084, -0.810836, 1.570796, 1.708247],accel_mss,speed_ms,0,blend_radius_m)
    |   movel([0.137003, -1.250600, -2.651014, -0.810775, 1.570796, 1.707799],accel_mss,speed_ms,0,blend_radius_m)
    |   movel([0.136737, -1.250566, -2.651032, -0.810791, 1.570796, 1.707533],accel_mss,speed_ms,0,blend_radius_m)
    |   movel([0.136577, -1.250358, -2.651143, -0.810888, 1.570796, 1.707374],accel_mss,speed_ms,0,blend_radius_m)
    |   movel([0.136485, -1.249888, -2.651394, -0.811107, 1.570796, 1.707281],accel_mss,speed_ms,0,blend_radius_m)
    |   movel([0.136093, -1.248988, -2.651874, -0.811527, 1.570796, 1.706889],accel_mss,speed_ms,0,blend_radius_m)
    |   movel([0.135259, -1.248595, -2.652083, -0.811711, 1.570796, 1.706056],accel_mss,speed_ms,0,blend_radius_m)
    |   movel([0.134232, -1.248815, -2.651966, -0.811608, 1.570796, 1.705028],accel_mss,speed_ms,0,blend_radius_m)
    |   movel([0.133293, -1.249559, -2.651569, -0.811260, 1.570796, 1.704090],accel_mss,speed_ms,0,blend_radius_m)
    |   movel([0.132861, -1.250341, -2.651152, -0.810896, 1.570796, 1.703657],accel_mss,speed_ms,0,blend_radius_m)
    |   movel([0.132871, -1.251012, -2.650794, -0.810583, 1.570796, 1.703667],accel_mss,speed_ms,0,blend_radius_m)
    |   movel([0.133354, -1.251468, -2.650550, -0.810371, 1.570796, 1.704151],accel_mss,speed_ms,0,blend_radius_m)
    |   movel([0.134238, -1.251642, -2.650456, -0.810290, 1.570796, 1.705035],accel_mss,speed_ms,0,blend_radius_m)
    |   movel([0.134548, -1.251641, -2.650457, -0.810291, 1.570796, 1.705344],accel_mss,speed_ms,0,blend_radius_m)
    |   movel([0.134854, -1.251627, -2.650465, -0.810298, 1.570796, 1.705650],accel_mss,speed_ms,0,blend_radius_m)
    |   movel([0.135274, -1.251568, -2.650496, -0.810325, 1.570796, 1.706071],accel_mss,speed_ms,0,blend_radius_m)
    |   movel([0.135532, -1.251584, -2.650487, -0.810317, 1.570796, 1.706328],accel_mss,speed_ms,0,blend_radius_m)
    |   movel([0.135756, -1.251751, -2.650398, -0.810240, 1.570796, 1.706552],accel_mss,speed_ms,0,blend_radius_m)
    |   movel([0.135846, -1.252036, -2.650246, -0.810108, 1.570796, 1.706642],accel_mss,speed_ms,0,blend_radius_m)
    |   movel([0.135832, -1.252571, -2.649958, -0.809860, 1.570796, 1.706628],accel_mss,speed_ms,0,blend_radius_m)
    |   movel([0.135724, -1.253517, -2.649450, -0.809422, 1.570796, 1.706520],accel_mss,speed_ms,0,blend_radius_m)
    |   movel([0.135420, -1.255572, -2.648342, -0.808475, 1.570796, 1.706217],accel_mss,speed_ms,0,blend_radius_m)
    |   movel([0.135034, -1.258058, -2.646995, -0.807336, 1.570796, 1.705830],accel_mss,speed_ms,0,blend_radius_m)
    |   movel([0.134814, -1.258982, -2.646492, -0.806914, 1.570796, 1.705611],accel_mss,speed_ms,0,blend_radius_m)
    |   movel([0.134542, -1.259451, -2.646237, -0.806701, 1.570796, 1.705338],accel_mss,speed_ms,0,blend_radius_m)
    |   movel([0.134131, -1.259731, -2.646084, -0.806574, 1.570796, 1.704927],accel_mss,speed_ms,0,blend_radius_m)
    |   movel([0.133824, -1.259748, -2.646075, -0.806566, 1.570796, 1.704620],accel_mss,speed_ms,0,blend_radius_m)
    |   movel([0.133658, -1.259591, -2.646161, -0.806637, 1.570796, 1.704454],accel_mss,speed_ms,0,blend_radius_m)
    |   movel([0.133614, -1.259182, -2.646384, -0.806824, 1.570796, 1.704411],accel_mss,speed_ms,0,blend_radius_m)
    |   movel([0.133693, -1.258313, -2.646857, -0.807220, 1.570796, 1.704489],accel_mss,speed_ms,0,blend_radius_m)
    |   movel([0.133760, -1.257672, -2.647205, -0.807512, 1.570796, 1.704556],accel_mss,speed_ms,0,blend_radius_m)
    |   movel([0.133768, -1.257296, -2.647409, -0.807684, 1.570796, 1.704565],accel_mss,speed_ms,0,blend_radius_m)
    |   movel([0.133641, -1.257005, -2.647567, -0.807817, 1.570796, 1.704437],accel_mss,speed_ms,0,blend_radius_m)
    |   movel([0.133135, -1.257023, -2.647557, -0.807809, 1.570796, 1.703932],accel_mss,speed_ms,0,blend_radius_m)
    |   movel([0.132693, -1.257059, -2.647538, -0.807793, 1.570796, 1.703489],accel_mss,speed_ms,0,blend_radius_m)
    |   movel([0.132205, -1.257107, -2.647512, -0.807771, 1.570796, 1.703001],accel_mss,speed_ms,0,blend_radius_m)
    |   movel([0.131165, -1.257148, -2.647489, -0.807752, 1.570796, 1.701961],accel_mss,speed_ms,0,blend_radius_m)
    |   movel([0.130280, -1.257046, -2.647545, -0.807799, 1.570796, 1.701076],accel_mss,speed_ms,0,blend_radius_m)
    |   movel([0.129498, -1.256778, -2.647690, -0.807922, 1.570796, 1.700295],accel_mss,speed_ms,0,blend_radius_m)
    |   movel([0.128756, -1.256342, -2.647926, -0.808121, 1.570796, 1.699553],accel_mss,speed_ms,0,blend_radius_m)
    |   movel([0.127629, -1.254975, -2.648665, -0.808749, 1.570796, 1.698425],accel_mss,speed_ms,0,blend_radius_m)
    |   movel([0.127239, -1.253124, -2.649661, -0.809604, 1.570796, 1.698036],accel_mss,speed_ms,0,blend_radius_m)
    |   movel([0.127630, -1.250874, -2.650868, -0.810648, 1.570796, 1.698426],accel_mss,speed_ms,0,blend_radius_m)
    |   movel([0.128781, -1.248347, -2.652215, -0.811827, 1.570796, 1.699577],accel_mss,speed_ms,0,blend_radius_m)
    |   movel([0.129174, -1.247712, -2.652552, -0.812125, 1.570796, 1.699970],accel_mss,speed_ms,0,blend_radius_m)
    |   movel([0.129602, -1.247109, -2.652872, -0.812408, 1.570796, 1.700398],accel_mss,speed_ms,0,blend_radius_m)
    |   movel([0.130119, -1.246465, -2.653213, -0.812710, 1.570796, 1.700916],accel_mss,speed_ms,0,blend_radius_m)
    |   movel([0.130785, -1.245709, -2.653613, -0.813066, 1.570796, 1.701581],accel_mss,speed_ms,0,blend_radius_m)
    |   movel([0.132478, -1.244039, -2.654494, -0.813856, 1.570796, 1.703274],accel_mss,speed_ms,0,blend_radius_m)
    |   movel([0.134231, -1.242693, -2.655202, -0.814494, 1.570796, 1.705028],accel_mss,speed_ms,0,blend_radius_m)
    |   movel([0.136117, -1.241632, -2.655759, -0.814999, 1.570796, 1.706913],accel_mss,speed_ms,0,blend_radius_m)
    |   movel([0.138201, -1.240803, -2.656192, -0.815394, 1.570796, 1.708998],accel_mss,speed_ms,0,blend_radius_m)
    |   movel([0.139435, -1.240437, -2.656383, -0.815568, 1.570796, 1.710232],accel_mss,speed_ms,0,blend_radius_m)
    |   movel([0.140458, -1.240212, -2.656501, -0.815676, 1.570796, 1.711255],accel_mss,speed_ms,0,blend_radius_m)
    |   movel([0.141377, -1.240102, -2.656558, -0.815729, 1.570796, 1.712174],accel_mss,speed_ms,0,blend_radius_m)
    |   movel([0.142291, -1.240094, -2.656562, -0.815732, 1.570796, 1.713088],accel_mss,speed_ms,0,blend_radius_m)
    |   movel([0.144324, -1.240459, -2.656372, -0.815558, 1.570796, 1.715120],accel_mss,speed_ms,0,blend_radius_m)
    |   movel([0.145972, -1.241324, -2.655920, -0.815145, 1.570796, 1.716769],accel_mss,speed_ms,0,blend_radius_m)
    |   movel([0.147123, -1.242616, -2.655243, -0.814531, 1.570796, 1.717920],accel_mss,speed_ms,0,blend_radius_m)
    |   movel([0.147683, -1.244233, -2.654392, -0.813764, 1.570796, 1.718479],accel_mss,speed_ms,0,blend_radius_m)
    |   movel([0.147706, -1.244999, -2.653988, -0.813402, 1.570796, 1.718502],accel_mss,speed_ms,0,blend_radius_m)
    |   movel([0.147581, -1.246087, -2.653414, -0.812888, 1.570796, 1.718377],accel_mss,speed_ms,0,blend_radius_m)
    |   movel([0.147363, -1.247199, -2.652824, -0.812365, 1.570796, 1.718159],accel_mss,speed_ms,0,blend_radius_m)
    |   movel([0.147089, -1.248042, -2.652377, -0.811970, 1.570796, 1.717886],accel_mss,speed_ms,0,blend_radius_m)
    |   movel([0.145883, -1.250181, -2.651238, -0.810970, 1.570796, 1.716679],accel_mss,speed_ms,0,blend_radius_m)
    |   movel([0.144114, -1.252178, -2.650169, -0.810042, 1.570796, 1.714911],accel_mss,speed_ms,0,blend_radius_m)
    |   movel([0.142022, -1.253780, -2.649308, -0.809300, 1.570796, 1.712819],accel_mss,speed_ms,0,blend_radius_m)
    |   movel([0.139874, -1.254782, -2.648769, -0.808838, 1.570796, 1.710670],accel_mss,speed_ms,0,blend_radius_m)
    |   movel([0.139347, -1.254993, -2.648655, -0.808741, 1.570796, 1.710143],accel_mss,speed_ms,0,blend_radius_m)
    |   movel([0.139026, -1.255205, -2.648540, -0.808644, 1.570796, 1.709822],accel_mss,speed_ms,0,blend_radius_m)
    |   movel([0.138790, -1.255798, -2.648220, -0.808371, 1.570796, 1.709586],accel_mss,speed_ms,0,blend_radius_m)
    |   movel([0.138626, -1.256330, -2.647932, -0.808127, 1.570796, 1.709423],accel_mss,speed_ms,0,blend_radius_m)
    |   movel([0.138465, -1.256921, -2.647612, -0.807856, 1.570796, 1.709261],accel_mss,speed_ms,0,blend_radius_m)
    |   movel([0.138304, -1.257512, -2.647292, -0.807586, 1.570796, 1.709100],accel_mss,speed_ms,0,blend_radius_m)
    |   movel([0.138138, -1.258043, -2.647003, -0.807343, 1.570796, 1.708934],accel_mss,speed_ms,0,blend_radius_m)
    |   movel([0.137986, -1.258487, -2.646762, -0.807140, 1.570796, 1.708782],accel_mss,speed_ms,0,blend_radius_m)
    |   movel([0.137718, -1.258809, -2.646587, -0.806993, 1.570796, 1.708514],accel_mss,speed_ms,0,blend_radius_m)
    |   movel([0.137358, -1.258904, -2.646535, -0.806950, 1.570796, 1.708154],accel_mss,speed_ms,0,blend_radius_m)
    |   speed_ms = 0.003
    |   movel([0.137358, -1.262485, -2.648225, -0.801679, 1.570796, 1.708154],accel_mss,speed_ms,0,blend_radius_m)
    |   speed_ms = 0.007
    |   movel([0.137144, -1.262197, -2.648383, -0.801809, 1.570796, 1.707940],accel_mss,speed_ms,0,blend_radius_m)
    |   movel([0.137235, -1.261543, -2.648740, -0.802106, 1.570796, 1.708031],accel_mss,speed_ms,0,blend_radius_m)
    |   movel([0.137436, -1.260465, -2.649328, -0.802596, 1.570796, 1.708233],accel_mss,speed_ms,0,blend_radius_m)
    |   movel([0.137871, -1.258394, -2.650453, -0.803542, 1.570796, 1.708667],accel_mss,speed_ms,0,blend_radius_m)
    |   movel([0.138200, -1.256898, -2.651263, -0.804228, 1.570796, 1.708997],accel_mss,speed_ms,0,blend_radius_m)
    |   movel([0.138501, -1.255609, -2.651959, -0.804821, 1.570796, 1.709297],accel_mss,speed_ms,0,blend_radius_m)
    |   movel([0.138778, -1.254482, -2.652565, -0.805342, 1.570796, 1.709574],accel_mss,speed_ms,0,blend_radius_m)
    |   movel([0.139175, -1.254068, -2.652788, -0.805533, 1.570796, 1.709971],accel_mss,speed_ms,0,blend_radius_m)
    |   movel([0.139446, -1.253850, -2.652904, -0.805634, 1.570796, 1.710242],accel_mss,speed_ms,0,blend_radius_m)
    |   movel([0.139737, -1.253627, -2.653024, -0.805738, 1.570796, 1.710534],accel_mss,speed_ms,0,blend_radius_m)
    |   movel([0.140340, -1.253121, -2.653295, -0.805972, 1.570796, 1.711136],accel_mss,speed_ms,0,blend_radius_m)
    |   movel([0.140778, -1.252648, -2.653549, -0.806192, 1.570796, 1.711574],accel_mss,speed_ms,0,blend_radius_m)
    |   movel([0.141088, -1.252162, -2.653809, -0.806418, 1.570796, 1.711885],accel_mss,speed_ms,0,blend_radius_m)
    |   movel([0.141299, -1.251625, -2.654096, -0.806668, 1.570796, 1.712095],accel_mss,speed_ms,0,blend_radius_m)
    |   movel([0.141376, -1.251288, -2.654276, -0.806825, 1.570796, 1.712172],accel_mss,speed_ms,0,blend_radius_m)
    |   movel([0.141270, -1.250932, -2.654465, -0.806991, 1.570796, 1.712067],accel_mss,speed_ms,0,blend_radius_m)
    |   movel([0.141024, -1.250736, -2.654570, -0.807083, 1.570796, 1.711820],accel_mss,speed_ms,0,blend_radius_m)
    |   movel([0.140322, -1.250541, -2.654674, -0.807174, 1.570796, 1.711118],accel_mss,speed_ms,0,blend_radius_m)
    |   movel([0.139577, -1.250824, -2.654523, -0.807042, 1.570796, 1.710374],accel_mss,speed_ms,0,blend_radius_m)
    |   movel([0.138926, -1.251547, -2.654137, -0.806704, 1.570796, 1.709723],accel_mss,speed_ms,0,blend_radius_m)
    |   movel([0.138497, -1.252583, -2.653584, -0.806223, 1.570796, 1.709294],accel_mss,speed_ms,0,blend_radius_m)
    |   movel([0.138299, -1.253267, -2.653217, -0.805905, 1.570796, 1.709096],accel_mss,speed_ms,0,blend_radius_m)
    |   movel([0.138115, -1.253625, -2.653026, -0.805739, 1.570796, 1.708911],accel_mss,speed_ms,0,blend_radius_m)
    |   movel([0.137451, -1.254066, -2.652789, -0.805534, 1.570796, 1.708247],accel_mss,speed_ms,0,blend_radius_m)
    |   movel([0.137003, -1.254196, -2.652719, -0.805474, 1.570796, 1.707799],accel_mss,speed_ms,0,blend_radius_m)
    |   movel([0.136737, -1.254162, -2.652737, -0.805490, 1.570796, 1.707533],accel_mss,speed_ms,0,blend_radius_m)
    |   movel([0.136577, -1.253955, -2.652848, -0.805586, 1.570796, 1.707374],accel_mss,speed_ms,0,blend_radius_m)
    |   movel([0.136485, -1.253486, -2.653100, -0.805803, 1.570796, 1.707281],accel_mss,speed_ms,0,blend_radius_m)
    |   movel([0.136093, -1.252587, -2.653581, -0.806221, 1.570796, 1.706889],accel_mss,speed_ms,0,blend_radius_m)
    |   movel([0.135259, -1.252195, -2.653791, -0.806403, 1.570796, 1.706056],accel_mss,speed_ms,0,blend_radius_m)
    |   movel([0.134232, -1.252414, -2.653674, -0.806301, 1.570796, 1.705028],accel_mss,speed_ms,0,blend_radius_m)
    |   movel([0.133293, -1.253158, -2.653276, -0.805956, 1.570796, 1.704090],accel_mss,speed_ms,0,blend_radius_m)
    |   movel([0.132861, -1.253938, -2.652858, -0.805594, 1.570796, 1.703657],accel_mss,speed_ms,0,blend_radius_m)
    |   movel([0.132871, -1.254607, -2.652498, -0.805284, 1.570796, 1.703667],accel_mss,speed_ms,0,blend_radius_m)
    |   movel([0.133354, -1.255063, -2.652253, -0.805073, 1.570796, 1.704151],accel_mss,speed_ms,0,blend_radius_m)
    |   movel([0.134238, -1.255236, -2.652159, -0.804993, 1.570796, 1.705035],accel_mss,speed_ms,0,blend_radius_m)
    |   movel([0.134548, -1.255236, -2.652160, -0.804994, 1.570796, 1.705344],accel_mss,speed_ms,0,blend_radius_m)
    |   movel([0.134854, -1.255221, -2.652168, -0.805000, 1.570796, 1.705650],accel_mss,speed_ms,0,blend_radius_m)
    |   movel([0.135274, -1.255162, -2.652199, -0.805027, 1.570796, 1.706071],accel_mss,speed_ms,0,blend_radius_m)
    |   movel([0.135532, -1.255179, -2.652190, -0.805020, 1.570796, 1.706328],accel_mss,speed_ms,0,blend_radius_m)
    |   movel([0.135756, -1.255345, -2.652101, -0.804943, 1.570796, 1.706552],accel_mss,speed_ms,0,blend_radius_m)
    |   movel([0.135846, -1.255629, -2.651948, -0.804812, 1.570796, 1.706642],accel_mss,speed_ms,0,blend_radius_m)
    |   movel([0.135832, -1.256164, -2.651660, -0.804566, 1.570796, 1.706628],accel_mss,speed_ms,0,blend_radius_m)
    |   movel([0.135724, -1.257108, -2.651150, -0.804131, 1.570796, 1.706520],accel_mss,speed_ms,0,blend_radius_m)
    |   movel([0.135420, -1.259159, -2.650038, -0.803192, 1.570796, 1.706217],accel_mss,speed_ms,0,blend_radius_m)
    |   movel([0.135034, -1.261640, -2.648687, -0.802062, 1.570796, 1.705830],accel_mss,speed_ms,0,blend_radius_m)
    |   movel([0.134814, -1.262562, -2.648183, -0.801644, 1.570796, 1.705611],accel_mss,speed_ms,0,blend_radius_m)
    |   movel([0.134542, -1.263030, -2.647926, -0.801432, 1.570796, 1.705338],accel_mss,speed_ms,0,blend_radius_m)
    |   movel([0.134131, -1.263310, -2.647773, -0.801306, 1.570796, 1.704927],accel_mss,speed_ms,0,blend_radius_m)
    |   movel([0.133824, -1.263327, -2.647764, -0.801298, 1.570796, 1.704620],accel_mss,speed_ms,0,blend_radius_m)
    |   movel([0.133658, -1.263170, -2.647850, -0.801369, 1.570796, 1.704454],accel_mss,speed_ms,0,blend_radius_m)
    |   movel([0.133614, -1.262762, -2.648074, -0.801554, 1.570796, 1.704411],accel_mss,speed_ms,0,blend_radius_m)
    |   movel([0.133693, -1.261894, -2.648548, -0.801946, 1.570796, 1.704489],accel_mss,speed_ms,0,blend_radius_m)
    |   movel([0.133760, -1.261255, -2.648897, -0.802237, 1.570796, 1.704556],accel_mss,speed_ms,0,blend_radius_m)
    |   movel([0.133768, -1.260879, -2.649102, -0.802408, 1.570796, 1.704565],accel_mss,speed_ms,0,blend_radius_m)
    |   movel([0.133641, -1.260589, -2.649260, -0.802540, 1.570796, 1.704437],accel_mss,speed_ms,0,blend_radius_m)
    |   movel([0.133135, -1.260607, -2.649251, -0.802531, 1.570796, 1.703932],accel_mss,speed_ms,0,blend_radius_m)
    |   movel([0.132693, -1.260643, -2.649231, -0.802515, 1.570796, 1.703489],accel_mss,speed_ms,0,blend_radius_m)
    |   movel([0.132205, -1.260691, -2.649205, -0.802493, 1.570796, 1.703001],accel_mss,speed_ms,0,blend_radius_m)
    |   movel([0.131165, -1.260732, -2.649182, -0.802474, 1.570796, 1.701961],accel_mss,speed_ms,0,blend_radius_m)
    |   movel([0.130280, -1.260630, -2.649238, -0.802521, 1.570796, 1.701076],accel_mss,speed_ms,0,blend_radius_m)
    |   movel([0.129498, -1.260362, -2.649384, -0.802643, 1.570796, 1.700295],accel_mss,speed_ms,0,blend_radius_m)
    |   movel([0.128756, -1.259927, -2.649621, -0.802841, 1.570796, 1.699553],accel_mss,speed_ms,0,blend_radius_m)
    |   movel([0.127629, -1.258563, -2.650362, -0.803464, 1.570796, 1.698425],accel_mss,speed_ms,0,blend_radius_m)
    |   movel([0.127239, -1.256715, -2.651362, -0.804312, 1.570796, 1.698036],accel_mss,speed_ms,0,blend_radius_m)
    |   movel([0.127630, -1.254470, -2.652572, -0.805348, 1.570796, 1.698426],accel_mss,speed_ms,0,blend_radius_m)
    |   movel([0.128781, -1.251947, -2.653924, -0.806518, 1.570796, 1.699577],accel_mss,speed_ms,0,blend_radius_m)
    |   movel([0.129174, -1.251314, -2.654262, -0.806813, 1.570796, 1.699970],accel_mss,speed_ms,0,blend_radius_m)
    |   movel([0.129602, -1.250711, -2.654583, -0.807095, 1.570796, 1.700398],accel_mss,speed_ms,0,blend_radius_m)
    |   movel([0.130119, -1.250069, -2.654925, -0.807395, 1.570796, 1.700916],accel_mss,speed_ms,0,blend_radius_m)
    |   movel([0.130785, -1.249315, -2.655326, -0.807748, 1.570796, 1.701581],accel_mss,speed_ms,0,blend_radius_m)
    |   movel([0.132478, -1.247647, -2.656210, -0.808531, 1.570796, 1.703274],accel_mss,speed_ms,0,blend_radius_m)
    |   movel([0.134231, -1.246303, -2.656921, -0.809165, 1.570796, 1.705028],accel_mss,speed_ms,0,blend_radius_m)
    |   movel([0.136117, -1.245244, -2.657479, -0.809666, 1.570796, 1.706913],accel_mss,speed_ms,0,blend_radius_m)
    |   movel([0.138201, -1.244417, -2.657914, -0.810058, 1.570796, 1.708998],accel_mss,speed_ms,0,blend_radius_m)
    |   movel([0.139435, -1.244052, -2.658105, -0.810232, 1.570796, 1.710232],accel_mss,speed_ms,0,blend_radius_m)
    |   movel([0.140458, -1.243828, -2.658223, -0.810338, 1.570796, 1.711255],accel_mss,speed_ms,0,blend_radius_m)
    |   movel([0.141377, -1.243717, -2.658281, -0.810391, 1.570796, 1.712174],accel_mss,speed_ms,0,blend_radius_m)
    |   movel([0.142291, -1.243709, -2.658285, -0.810394, 1.570796, 1.713088],accel_mss,speed_ms,0,blend_radius_m)
    |   movel([0.144324, -1.244073, -2.658094, -0.810221, 1.570796, 1.715120],accel_mss,speed_ms,0,blend_radius_m)
    |   movel([0.145972, -1.244937, -2.657640, -0.809811, 1.570796, 1.716769],accel_mss,speed_ms,0,blend_radius_m)
    |   movel([0.147123, -1.246227, -2.656961, -0.809201, 1.570796, 1.717920],accel_mss,speed_ms,0,blend_radius_m)
    |   movel([0.147683, -1.247841, -2.656108, -0.808440, 1.570796, 1.718479],accel_mss,speed_ms,0,blend_radius_m)
    |   movel([0.147706, -1.248606, -2.655703, -0.808081, 1.570796, 1.718502],accel_mss,speed_ms,0,blend_radius_m)
    |   movel([0.147581, -1.249692, -2.655126, -0.807572, 1.570796, 1.718377],accel_mss,speed_ms,0,blend_radius_m)
    |   movel([0.147363, -1.250802, -2.654535, -0.807052, 1.570796, 1.718159],accel_mss,speed_ms,0,blend_radius_m)
    |   movel([0.147089, -1.251643, -2.654086, -0.806660, 1.570796, 1.717886],accel_mss,speed_ms,0,blend_radius_m)
    |   movel([0.145883, -1.253778, -2.652943, -0.805668, 1.570796, 1.716679],accel_mss,speed_ms,0,blend_radius_m)
    |   movel([0.144114, -1.255772, -2.651871, -0.804746, 1.570796, 1.714911],accel_mss,speed_ms,0,blend_radius_m)
    |   movel([0.142022, -1.257371, -2.651008, -0.804011, 1.570796, 1.712819],accel_mss,speed_ms,0,blend_radius_m)
    |   movel([0.139874, -1.258370, -2.650466, -0.803552, 1.570796, 1.710670],accel_mss,speed_ms,0,blend_radius_m)
    |   movel([0.139347, -1.258581, -2.650352, -0.803456, 1.570796, 1.710143],accel_mss,speed_ms,0,blend_radius_m)
    |   movel([0.139026, -1.258793, -2.650237, -0.803359, 1.570796, 1.709822],accel_mss,speed_ms,0,blend_radius_m)
    |   movel([0.138790, -1.259384, -2.649916, -0.803089, 1.570796, 1.709586],accel_mss,speed_ms,0,blend_radius_m)
    |   movel([0.138626, -1.259915, -2.649627, -0.802847, 1.570796, 1.709423],accel_mss,speed_ms,0,blend_radius_m)
    |   movel([0.138465, -1.260505, -2.649306, -0.802578, 1.570796, 1.709261],accel_mss,speed_ms,0,blend_radius_m)
    |   movel([0.138304, -1.261095, -2.648985, -0.802310, 1.570796, 1.709100],accel_mss,speed_ms,0,blend_radius_m)
    |   movel([0.138138, -1.261625, -2.648695, -0.802069, 1.570796, 1.708934],accel_mss,speed_ms,0,blend_radius_m)
    |   movel([0.137986, -1.262068, -2.648453, -0.801868, 1.570796, 1.708782],accel_mss,speed_ms,0,blend_radius_m)
    |   movel([0.137718, -1.262390, -2.648277, -0.801722, 1.570796, 1.708514],accel_mss,speed_ms,0,blend_radius_m)
    |   movel([0.137358, -1.262485, -2.648225, -0.801679, 1.570796, 1.708154],accel_mss,speed_ms,0,blend_radius_m)
    |   speed_ms = 0.003
    |   movel([0.137358, -1.248347, -2.641414, -0.822628, 1.570796, 1.708154],accel_mss,speed_ms,0,blend_radius_m)
    |   speed_ms = 1.000
    |   movel([0.137358, -1.221519, -2.627413, -0.863457, 1.570796, 1.708154],accel_mss,speed_ms,0,blend_radius_m)
    |   movel([0.136331, -1.221369, -2.627491, -0.863529, 1.570796, 1.707127],accel_mss,speed_ms,0,blend_radius_m)
    |   movel([0.136331, -1.248198, -2.641494, -0.822697, 1.570796, 1.707127],accel_mss,speed_ms,0,blend_radius_m)
    |   speed_ms = 0.003
    |   movel([0.136331, -1.258756, -2.646615, -0.807017, 1.570796, 1.707127],accel_mss,speed_ms,0,blend_radius_m)
    |   speed_ms = 0.007
    |   movel([0.135965, -1.259022, -2.646471, -0.806896, 1.570796, 1.706761],accel_mss,speed_ms,0,blend_radius_m)
    |   movel([0.135639, -1.258950, -2.646510, -0.806929, 1.570796, 1.706435],accel_mss,speed_ms,0,blend_radius_m)
    |   movel([0.135615, -1.258574, -2.646715, -0.807101, 1.570796, 1.706412],accel_mss,speed_ms,0,blend_radius_m)
    |   movel([0.136097, -1.255221, -2.648532, -0.808636, 1.570796, 1.706894],accel_mss,speed_ms,0,blend_radius_m)
    |   movel([0.136603, -1.251789, -2.650378, -0.810222, 1.570796, 1.707400],accel_mss,speed_ms,0,blend_radius_m)
    |   movel([0.136724, -1.251497, -2.650534, -0.810358, 1.570796, 1.707521],accel_mss,speed_ms,0,blend_radius_m)
    |   movel([0.137247, -1.251196, -2.650695, -0.810498, 1.570796, 1.708044],accel_mss,speed_ms,0,blend_radius_m)
    |   movel([0.137587, -1.251126, -2.650733, -0.810530, 1.570796, 1.708383],accel_mss,speed_ms,0,blend_radius_m)
    |   movel([0.137884, -1.251389, -2.650592, -0.810408, 1.570796, 1.708680],accel_mss,speed_ms,0,blend_radius_m)
    |   movel([0.137821, -1.251968, -2.650282, -0.810139, 1.570796, 1.708618],accel_mss,speed_ms,0,blend_radius_m)
    |   movel([0.137622, -1.253027, -2.649713, -0.809648, 1.570796, 1.708419],accel_mss,speed_ms,0,blend_radius_m)
    |   movel([0.137096, -1.255476, -2.648394, -0.808519, 1.570796, 1.707892],accel_mss,speed_ms,0,blend_radius_m)
    |   movel([0.136830, -1.256677, -2.647744, -0.807968, 1.570796, 1.707626],accel_mss,speed_ms,0,blend_radius_m)
    |   movel([0.136591, -1.257717, -2.647180, -0.807492, 1.570796, 1.707388],accel_mss,speed_ms,0,blend_radius_m)
    |   movel([0.136382, -1.258618, -2.646691, -0.807081, 1.570796, 1.707178],accel_mss,speed_ms,0,blend_radius_m)
    |   speed_ms = 0.003
    |   movel([0.136331, -1.262337, -2.648306, -0.801746, 1.570796, 1.707127],accel_mss,speed_ms,0,blend_radius_m)
    |   speed_ms = 0.007
    |   movel([0.135965, -1.262602, -2.648161, -0.801626, 1.570796, 1.706761],accel_mss,speed_ms,0,blend_radius_m)
    |   movel([0.135639, -1.262530, -2.648201, -0.801659, 1.570796, 1.706435],accel_mss,speed_ms,0,blend_radius_m)
    |   movel([0.135615, -1.262155, -2.648406, -0.801828, 1.570796, 1.706412],accel_mss,speed_ms,0,blend_radius_m)
    |   movel([0.136097, -1.258809, -2.650228, -0.803352, 1.570796, 1.706894],accel_mss,speed_ms,0,blend_radius_m)
    |   movel([0.136603, -1.255383, -2.652081, -0.804926, 1.570796, 1.707400],accel_mss,speed_ms,0,blend_radius_m)
    |   movel([0.136724, -1.255092, -2.652237, -0.805060, 1.570796, 1.707521],accel_mss,speed_ms,0,blend_radius_m)
    |   movel([0.137247, -1.254791, -2.652399, -0.805199, 1.570796, 1.708044],accel_mss,speed_ms,0,blend_radius_m)
    |   movel([0.137587, -1.254721, -2.652437, -0.805231, 1.570796, 1.708383],accel_mss,speed_ms,0,blend_radius_m)
    |   movel([0.137884, -1.254983, -2.652296, -0.805110, 1.570796, 1.708680],accel_mss,speed_ms,0,blend_radius_m)
    |   movel([0.137821, -1.255562, -2.651984, -0.804843, 1.570796, 1.708618],accel_mss,speed_ms,0,blend_radius_m)
    |   movel([0.137622, -1.256619, -2.651414, -0.804356, 1.570796, 1.708419],accel_mss,speed_ms,0,blend_radius_m)
    |   movel([0.137096, -1.259063, -2.650090, -0.803235, 1.570796, 1.707892],accel_mss,speed_ms,0,blend_radius_m)
    |   movel([0.136830, -1.260262, -2.649439, -0.802689, 1.570796, 1.707626],accel_mss,speed_ms,0,blend_radius_m)
    |   movel([0.136591, -1.261299, -2.648873, -0.802217, 1.570796, 1.707388],accel_mss,speed_ms,0,blend_radius_m)
    |   movel([0.136382, -1.262199, -2.648382, -0.801809, 1.570796, 1.707178],accel_mss,speed_ms,0,blend_radius_m)
    |   speed_ms = 0.003
    |   movel([0.136331, -1.248198, -2.641494, -0.822697, 1.570796, 1.707127],accel_mss,speed_ms,0,blend_radius_m)
    |   speed_ms = 1.000
    |   movel([0.136331, -1.221369, -2.627491, -0.863529, 1.570796, 1.707127],accel_mss,speed_ms,0,blend_radius_m)
    |   movel([0.135518, -1.213284, -2.631635, -0.867470, 1.570796, 1.706315],accel_mss,speed_ms,0,blend_radius_m)
    |   movel([0.135518, -1.240201, -2.645745, -0.826443, 1.570796, 1.706315],accel_mss,speed_ms,0,blend_radius_m)
    |   speed_ms = 0.003
    |   movel([0.135518, -1.250801, -2.650907, -0.810681, 1.570796, 1.706315],accel_mss,speed_ms,0,blend_radius_m)
    |   speed_ms = 0.007
    |   movel([0.135184, -1.250928, -2.650838, -0.810622, 1.570796, 1.705981],accel_mss,speed_ms,0,blend_radius_m)
    |   movel([0.134896, -1.250953, -2.650826, -0.810611, 1.570796, 1.705692],accel_mss,speed_ms,0,blend_radius_m)
    |   movel([0.134573, -1.250950, -2.650827, -0.810612, 1.570796, 1.705369],accel_mss,speed_ms,0,blend_radius_m)
    |   movel([0.134262, -1.250915, -2.650845, -0.810628, 1.570796, 1.705059],accel_mss,speed_ms,0,blend_radius_m)
    |   movel([0.133875, -1.250842, -2.650884, -0.810662, 1.570796, 1.704671],accel_mss,speed_ms,0,blend_radius_m)
    |   movel([0.133663, -1.250756, -2.650931, -0.810702, 1.570796, 1.704460],accel_mss,speed_ms,0,blend_radius_m)
    |   movel([0.133527, -1.250440, -2.651099, -0.810849, 1.570796, 1.704323],accel_mss,speed_ms,0,blend_radius_m)
    |   movel([0.133693, -1.249935, -2.651369, -0.811085, 1.570796, 1.704489],accel_mss,speed_ms,0,blend_radius_m)
    |   movel([0.134107, -1.249492, -2.651605, -0.811291, 1.570796, 1.704903],accel_mss,speed_ms,0,blend_radius_m)
    |   movel([0.134658, -1.249246, -2.651736, -0.811407, 1.570796, 1.705455],accel_mss,speed_ms,0,blend_radius_m)
    |   movel([0.135181, -1.249271, -2.651723, -0.811395, 1.570796, 1.705978],accel_mss,speed_ms,0,blend_radius_m)
    |   movel([0.135427, -1.249443, -2.651631, -0.811314, 1.570796, 1.706223],accel_mss,speed_ms,0,blend_radius_m)
    |   movel([0.135661, -1.249807, -2.651437, -0.811145, 1.570796, 1.706457],accel_mss,speed_ms,0,blend_radius_m)
    |   movel([0.135822, -1.250215, -2.651220, -0.810954, 1.570796, 1.706618],accel_mss,speed_ms,0,blend_radius_m)
    |   movel([0.135808, -1.250511, -2.651062, -0.810817, 1.570796, 1.706604],accel_mss,speed_ms,0,blend_radius_m)
    |   movel([0.135518, -1.250801, -2.650907, -0.810681, 1.570796, 1.706315],accel_mss,speed_ms,0,blend_radius_m)
    |   speed_ms = 0.003
    |   movel([0.135518, -1.254397, -2.652611, -0.805381, 1.570796, 1.706315],accel_mss,speed_ms,0,blend_radius_m)
    |   speed_ms = 0.007
    |   movel([0.135184, -1.254524, -2.652543, -0.805322, 1.570796, 1.705981],accel_mss,speed_ms,0,blend_radius_m)
    |   movel([0.134896, -1.254548, -2.652530, -0.805311, 1.570796, 1.705692],accel_mss,speed_ms,0,blend_radius_m)
    |   movel([0.134573, -1.254545, -2.652531, -0.805312, 1.570796, 1.705369],accel_mss,speed_ms,0,blend_radius_m)
    |   movel([0.134262, -1.254511, -2.652550, -0.805328, 1.570796, 1.705059],accel_mss,speed_ms,0,blend_radius_m)
    |   movel([0.133875, -1.254438, -2.652589, -0.805362, 1.570796, 1.704671],accel_mss,speed_ms,0,blend_radius_m)
    |   movel([0.133663, -1.254352, -2.652635, -0.805402, 1.570796, 1.704460],accel_mss,speed_ms,0,blend_radius_m)
    |   movel([0.133527, -1.254037, -2.652804, -0.805548, 1.570796, 1.704323],accel_mss,speed_ms,0,blend_radius_m)
    |   movel([0.133693, -1.253533, -2.653075, -0.805781, 1.570796, 1.704489],accel_mss,speed_ms,0,blend_radius_m)
    |   movel([0.134107, -1.253091, -2.653312, -0.805987, 1.570796, 1.704903],accel_mss,speed_ms,0,blend_radius_m)
    |   movel([0.134658, -1.252845, -2.653444, -0.806101, 1.570796, 1.705455],accel_mss,speed_ms,0,blend_radius_m)
    |   movel([0.135181, -1.252869, -2.653430, -0.806089, 1.570796, 1.705978],accel_mss,speed_ms,0,blend_radius_m)
    |   movel([0.135427, -1.253041, -2.653338, -0.806009, 1.570796, 1.706223],accel_mss,speed_ms,0,blend_radius_m)
    |   movel([0.135661, -1.253405, -2.653143, -0.805841, 1.570796, 1.706457],accel_mss,speed_ms,0,blend_radius_m)
    |   movel([0.135822, -1.253812, -2.652925, -0.805652, 1.570796, 1.706618],accel_mss,speed_ms,0,blend_radius_m)
    |   movel([0.135808, -1.254107, -2.652767, -0.805515, 1.570796, 1.706604],accel_mss,speed_ms,0,blend_radius_m)
    |   movel([0.135518, -1.254397, -2.652611, -0.805381, 1.570796, 1.706315],accel_mss,speed_ms,0,blend_radius_m)
    |   speed_ms = 0.003
    |   movel([0.135518, -1.240201, -2.645745, -0.826443, 1.570796, 1.706315],accel_mss,speed_ms,0,blend_radius_m)
    |   speed_ms = 1.000
    |   movel([0.135518, -1.213284, -2.631635, -0.867470, 1.570796, 1.706315],accel_mss,speed_ms,0,blend_radius_m)
    |   movel([0.139093, -1.211934, -2.632319, -0.868135, 1.570796, 1.709889],accel_mss,speed_ms,0,blend_radius_m)
    |   movel([0.139093, -1.238865, -2.646447, -0.827076, 1.570796, 1.709889],accel_mss,speed_ms,0,blend_radius_m)
    |   speed_ms = 0.003
    |   movel([0.139093, -1.249472, -2.651616, -0.811301, 1.570796, 1.709889],accel_mss,speed_ms,0,blend_radius_m)
    |   speed_ms = 0.007
    |   movel([0.139118, -1.249017, -2.651858, -0.811513, 1.570796, 1.709914],accel_mss,speed_ms,0,blend_radius_m)
    |   movel([0.139248, -1.248505, -2.652131, -0.811753, 1.570796, 1.710045],accel_mss,speed_ms,0,blend_radius_m)
    |   movel([0.139468, -1.248099, -2.652347, -0.811943, 1.570796, 1.710264],accel_mss,speed_ms,0,blend_radius_m)
    |   movel([0.139744, -1.247818, -2.652496, -0.812075, 1.570796, 1.710540],accel_mss,speed_ms,0,blend_radius_m)
    |   movel([0.140071, -1.247632, -2.652595, -0.812162, 1.570796, 1.710868],accel_mss,speed_ms,0,blend_radius_m)
    |   movel([0.140367, -1.247587, -2.652619, -0.812183, 1.570796, 1.711163],accel_mss,speed_ms,0,blend_radius_m)
    |   movel([0.140630, -1.247982, -2.652409, -0.811998, 1.570796, 1.711426],accel_mss,speed_ms,0,blend_radius_m)
    |   movel([0.140571, -1.248308, -2.652236, -0.811845, 1.570796, 1.711368],accel_mss,speed_ms,0,blend_radius_m)
    |   movel([0.140360, -1.248691, -2.652032, -0.811666, 1.570796, 1.711157],accel_mss,speed_ms,0,blend_radius_m)
    |   movel([0.139989, -1.249142, -2.651792, -0.811455, 1.570796, 1.710786],accel_mss,speed_ms,0,blend_radius_m)
    |   movel([0.139673, -1.249473, -2.651615, -0.811300, 1.570796, 1.710469],accel_mss,speed_ms,0,blend_radius_m)
    |   movel([0.139344, -1.249692, -2.651499, -0.811198, 1.570796, 1.710140],accel_mss,speed_ms,0,blend_radius_m)
    |   movel([0.139093, -1.249472, -2.651616, -0.811301, 1.570796, 1.709889],accel_mss,speed_ms,0,blend_radius_m)
    |   speed_ms = 0.003
    |   movel([0.139093, -1.253071, -2.653322, -0.805996, 1.570796, 1.709889],accel_mss,speed_ms,0,blend_radius_m)
    |   speed_ms = 0.007
    |   movel([0.139118, -1.252616, -2.653566, -0.806207, 1.570796, 1.709914],accel_mss,speed_ms,0,blend_radius_m)
    |   movel([0.139248, -1.252105, -2.653839, -0.806445, 1.570796, 1.710045],accel_mss,speed_ms,0,blend_radius_m)
    |   movel([0.139468, -1.251700, -2.654056, -0.806633, 1.570796, 1.710264],accel_mss,speed_ms,0,blend_radius_m)
    |   movel([0.139744, -1.251419, -2.654206, -0.806764, 1.570796, 1.710540],accel_mss,speed_ms,0,blend_radius_m)
    |   movel([0.140071, -1.251234, -2.654304, -0.806851, 1.570796, 1.710868],accel_mss,speed_ms,0,blend_radius_m)
    |   movel([0.140367, -1.251188, -2.654329, -0.806872, 1.570796, 1.711163],accel_mss,speed_ms,0,blend_radius_m)
    |   movel([0.140630, -1.251583, -2.654118, -0.806688, 1.570796, 1.711426],accel_mss,speed_ms,0,blend_radius_m)
    |   movel([0.140571, -1.251909, -2.653944, -0.806536, 1.570796, 1.711368],accel_mss,speed_ms,0,blend_radius_m)
    |   movel([0.140360, -1.252291, -2.653740, -0.806358, 1.570796, 1.711157],accel_mss,speed_ms,0,blend_radius_m)
    |   movel([0.139989, -1.252740, -2.653499, -0.806149, 1.570796, 1.710786],accel_mss,speed_ms,0,blend_radius_m)
    |   movel([0.139673, -1.253072, -2.653322, -0.805995, 1.570796, 1.710469],accel_mss,speed_ms,0,blend_radius_m)
    |   movel([0.139344, -1.253290, -2.653205, -0.805894, 1.570796, 1.710140],accel_mss,speed_ms,0,blend_radius_m)
    |   movel([0.139093, -1.253071, -2.653322, -0.805996, 1.570796, 1.709889],accel_mss,speed_ms,0,blend_radius_m)
    |   speed_ms = 0.003
    |   movel([0.139093, -1.238865, -2.646447, -0.827076, 1.570796, 1.709889],accel_mss,speed_ms,0,blend_radius_m)
    |   speed_ms = 1.000
    |   movel([0.139093, -1.211934, -2.632319, -0.868135, 1.570796, 1.709889],accel_mss,speed_ms,0,blend_radius_m)
    |   movel([0.082807, -1.213918, -2.631313, -0.867159, 1.570796, 1.653603],accel_mss,speed_ms,0,blend_radius_m)
    |   movel([0.082807, -1.240828, -2.645414, -0.826147, 1.570796, 1.653603],accel_mss,speed_ms,0,blend_radius_m)
    |   speed_ms = 0.003
    |   movel([0.082807, -1.251425, -2.650573, -0.810391, 1.570796, 1.653603],accel_mss,speed_ms,0,blend_radius_m)
    |   speed_ms = 0.007
    |   movel([0.081255, -1.253623, -2.649393, -0.809373, 1.570796, 1.652051],accel_mss,speed_ms,0,blend_radius_m)
    |   movel([0.079525, -1.256064, -2.648076, -0.808249, 1.570796, 1.650321],accel_mss,speed_ms,0,blend_radius_m)
    |   movel([0.077484, -1.258933, -2.646519, -0.806937, 1.570796, 1.648280],accel_mss,speed_ms,0,blend_radius_m)
    |   movel([0.074500, -1.263106, -2.644237, -0.805046, 1.570796, 1.645296],accel_mss,speed_ms,0,blend_radius_m)
    |   movel([0.072945, -1.265220, -2.643072, -0.804097, 1.570796, 1.643742],accel_mss,speed_ms,0,blend_radius_m)
    |   movel([0.072027, -1.266399, -2.642421, -0.803570, 1.570796, 1.642823],accel_mss,speed_ms,0,blend_radius_m)
    |   movel([0.072454, -1.264954, -2.643219, -0.804216, 1.570796, 1.643251],accel_mss,speed_ms,0,blend_radius_m)
    |   movel([0.073107, -1.263398, -2.644076, -0.804915, 1.570796, 1.643903],accel_mss,speed_ms,0,blend_radius_m)
    |   movel([0.073883, -1.261564, -2.645082, -0.805742, 1.570796, 1.644679],accel_mss,speed_ms,0,blend_radius_m)
    |   movel([0.074867, -1.259224, -2.646361, -0.806804, 1.570796, 1.645663],accel_mss,speed_ms,0,blend_radius_m)
    |   movel([0.075443, -1.257792, -2.647140, -0.807458, 1.570796, 1.646239],accel_mss,speed_ms,0,blend_radius_m)
    |   movel([0.075810, -1.256811, -2.647672, -0.807906, 1.570796, 1.646606],accel_mss,speed_ms,0,blend_radius_m)
    |   movel([0.075634, -1.256569, -2.647803, -0.808017, 1.570796, 1.646430],accel_mss,speed_ms,0,blend_radius_m)
    |   movel([0.075253, -1.256647, -2.647761, -0.807982, 1.570796, 1.646050],accel_mss,speed_ms,0,blend_radius_m)
    |   movel([0.074598, -1.256851, -2.647650, -0.807888, 1.570796, 1.645394],accel_mss,speed_ms,0,blend_radius_m)
    |   movel([0.073341, -1.257289, -2.647413, -0.807688, 1.570796, 1.644137],accel_mss,speed_ms,0,blend_radius_m)
    |   movel([0.072270, -1.257663, -2.647210, -0.807516, 1.570796, 1.643066],accel_mss,speed_ms,0,blend_radius_m)
    |   movel([0.071543, -1.257893, -2.647085, -0.807411, 1.570796, 1.642339],accel_mss,speed_ms,0,blend_radius_m)
    |   movel([0.071034, -1.258033, -2.647009, -0.807347, 1.570796, 1.641830],accel_mss,speed_ms,0,blend_radius_m)
    |   movel([0.070865, -1.257859, -2.647103, -0.807427, 1.570796, 1.641661],accel_mss,speed_ms,0,blend_radius_m)
    |   movel([0.071306, -1.256707, -2.647728, -0.807954, 1.570796, 1.642103],accel_mss,speed_ms,0,blend_radius_m)
    |   movel([0.071948, -1.255121, -2.648586, -0.808682, 1.570796, 1.642744],accel_mss,speed_ms,0,blend_radius_m)
    |   movel([0.072961, -1.252711, -2.649883, -0.809795, 1.570796, 1.643757],accel_mss,speed_ms,0,blend_radius_m)
    |   movel([0.073821, -1.250693, -2.650965, -0.810732, 1.570796, 1.644617],accel_mss,speed_ms,0,blend_radius_m)
    |   movel([0.074573, -1.248951, -2.651893, -0.811544, 1.570796, 1.645369],accel_mss,speed_ms,0,blend_radius_m)
    |   movel([0.075236, -1.247422, -2.652706, -0.812261, 1.570796, 1.646032],accel_mss,speed_ms,0,blend_radius_m)
    |   movel([0.075486, -1.247116, -2.652869, -0.812405, 1.570796, 1.646282],accel_mss,speed_ms,0,blend_radius_m)
    |   movel([0.076173, -1.246818, -2.653027, -0.812545, 1.570796, 1.646970],accel_mss,speed_ms,0,blend_radius_m)
    |   movel([0.077201, -1.246406, -2.653245, -0.812738, 1.570796, 1.647997],accel_mss,speed_ms,0,blend_radius_m)
    |   movel([0.078902, -1.245763, -2.653585, -0.813041, 1.570796, 1.649699],accel_mss,speed_ms,0,blend_radius_m)
    |   movel([0.080795, -1.245067, -2.653953, -0.813370, 1.570796, 1.651591],accel_mss,speed_ms,0,blend_radius_m)
    |   movel([0.081727, -1.244749, -2.654120, -0.813520, 1.570796, 1.652524],accel_mss,speed_ms,0,blend_radius_m)
    |   movel([0.082276, -1.244594, -2.654202, -0.813593, 1.570796, 1.653072],accel_mss,speed_ms,0,blend_radius_m)
    |   movel([0.082396, -1.244795, -2.654096, -0.813498, 1.570796, 1.653193],accel_mss,speed_ms,0,blend_radius_m)
    |   movel([0.081838, -1.245860, -2.653533, -0.812995, 1.570796, 1.652635],accel_mss,speed_ms,0,blend_radius_m)
    |   movel([0.081159, -1.247118, -2.652868, -0.812404, 1.570796, 1.651955],accel_mss,speed_ms,0,blend_radius_m)
    |   movel([0.080328, -1.248601, -2.652080, -0.811708, 1.570796, 1.651124],accel_mss,speed_ms,0,blend_radius_m)
    |   movel([0.079241, -1.250532, -2.651050, -0.810807, 1.570796, 1.650037],accel_mss,speed_ms,0,blend_radius_m)
    |   movel([0.078655, -1.251629, -2.650463, -0.810296, 1.570796, 1.649451],accel_mss,speed_ms,0,blend_radius_m)
    |   movel([0.078314, -1.252329, -2.650088, -0.809972, 1.570796, 1.649110],accel_mss,speed_ms,0,blend_radius_m)
    |   movel([0.078472, -1.252579, -2.649954, -0.809856, 1.570796, 1.649269],accel_mss,speed_ms,0,blend_radius_m)
    |   movel([0.078805, -1.252519, -2.649986, -0.809884, 1.570796, 1.649601],accel_mss,speed_ms,0,blend_radius_m)
    |   movel([0.079378, -1.252348, -2.650078, -0.809963, 1.570796, 1.650175],accel_mss,speed_ms,0,blend_radius_m)
    |   movel([0.080470, -1.251972, -2.650280, -0.810137, 1.570796, 1.651266],accel_mss,speed_ms,0,blend_radius_m)
    |   movel([0.081795, -1.251513, -2.650525, -0.810350, 1.570796, 1.652591],accel_mss,speed_ms,0,blend_radius_m)
    |   movel([0.082424, -1.251323, -2.650627, -0.810439, 1.570796, 1.653221],accel_mss,speed_ms,0,blend_radius_m)
    |   movel([0.082757, -1.251264, -2.650659, -0.810466, 1.570796, 1.653553],accel_mss,speed_ms,0,blend_radius_m)
    |   speed_ms = 0.003
    |   movel([0.082807, -1.255019, -2.652276, -0.805093, 1.570796, 1.653603],accel_mss,speed_ms,0,blend_radius_m)
    |   speed_ms = 0.007
    |   movel([0.081255, -1.257214, -2.651093, -0.804083, 1.570796, 1.652051],accel_mss,speed_ms,0,blend_radius_m)
    |   movel([0.079525, -1.259650, -2.649772, -0.802968, 1.570796, 1.650321],accel_mss,speed_ms,0,blend_radius_m)
    |   movel([0.077484, -1.262513, -2.648210, -0.801666, 1.570796, 1.648280],accel_mss,speed_ms,0,blend_radius_m)
    |   movel([0.074500, -1.266678, -2.645920, -0.799791, 1.570796, 1.645296],accel_mss,speed_ms,0,blend_radius_m)
    |   movel([0.072945, -1.268788, -2.644752, -0.798849, 1.570796, 1.643742],accel_mss,speed_ms,0,blend_radius_m)
    |   movel([0.072027, -1.269965, -2.644098, -0.798326, 1.570796, 1.642823],accel_mss,speed_ms,0,blend_radius_m)
    |   movel([0.072454, -1.268522, -2.644899, -0.798967, 1.570796, 1.643251],accel_mss,speed_ms,0,blend_radius_m)
    |   movel([0.073107, -1.266970, -2.645759, -0.799660, 1.570796, 1.643903],accel_mss,speed_ms,0,blend_radius_m)
    |   movel([0.073883, -1.265139, -2.646768, -0.800481, 1.570796, 1.644679],accel_mss,speed_ms,0,blend_radius_m)
    |   movel([0.074867, -1.262803, -2.648051, -0.801535, 1.570796, 1.645663],accel_mss,speed_ms,0,blend_radius_m)
    |   movel([0.075443, -1.261374, -2.648832, -0.802183, 1.570796, 1.646239],accel_mss,speed_ms,0,blend_radius_m)
    |   movel([0.075810, -1.260395, -2.649366, -0.802628, 1.570796, 1.646606],accel_mss,speed_ms,0,blend_radius_m)
    |   movel([0.075634, -1.260153, -2.649498, -0.802738, 1.570796, 1.646430],accel_mss,speed_ms,0,blend_radius_m)
    |   movel([0.075253, -1.260231, -2.649455, -0.802702, 1.570796, 1.646050],accel_mss,speed_ms,0,blend_radius_m)
    |   movel([0.074598, -1.260436, -2.649344, -0.802609, 1.570796, 1.645394],accel_mss,speed_ms,0,blend_radius_m)
    |   movel([0.073341, -1.260872, -2.649106, -0.802411, 1.570796, 1.644137],accel_mss,speed_ms,0,blend_radius_m)
    |   movel([0.072270, -1.261246, -2.648902, -0.802241, 1.570796, 1.643066],accel_mss,speed_ms,0,blend_radius_m)
    |   movel([0.071543, -1.261476, -2.648777, -0.802136, 1.570796, 1.642339],accel_mss,speed_ms,0,blend_radius_m)
    |   movel([0.071034, -1.261615, -2.648701, -0.802073, 1.570796, 1.641830],accel_mss,speed_ms,0,blend_radius_m)
    |   movel([0.070865, -1.261441, -2.648796, -0.802152, 1.570796, 1.641661],accel_mss,speed_ms,0,blend_radius_m)
    |   movel([0.071306, -1.260292, -2.649422, -0.802675, 1.570796, 1.642103],accel_mss,speed_ms,0,blend_radius_m)
    |   movel([0.071948, -1.258709, -2.650283, -0.803397, 1.570796, 1.642744],accel_mss,speed_ms,0,blend_radius_m)
    |   movel([0.072961, -1.256303, -2.651584, -0.804501, 1.570796, 1.643757],accel_mss,speed_ms,0,blend_radius_m)
    |   movel([0.073821, -1.254289, -2.652669, -0.805431, 1.570796, 1.644617],accel_mss,speed_ms,0,blend_radius_m)
    |   movel([0.074573, -1.252551, -2.653601, -0.806237, 1.570796, 1.645369],accel_mss,speed_ms,0,blend_radius_m)
    |   movel([0.075236, -1.251024, -2.654416, -0.806948, 1.570796, 1.646032],accel_mss,speed_ms,0,blend_radius_m)
    |   movel([0.075486, -1.250718, -2.654579, -0.807091, 1.570796, 1.646282],accel_mss,speed_ms,0,blend_radius_m)
    |   movel([0.076173, -1.250421, -2.654738, -0.807230, 1.570796, 1.646970],accel_mss,speed_ms,0,blend_radius_m)
    |   movel([0.077201, -1.250010, -2.654957, -0.807423, 1.570796, 1.647997],accel_mss,speed_ms,0,blend_radius_m)
    |   movel([0.078902, -1.249368, -2.655298, -0.807723, 1.570796, 1.649699],accel_mss,speed_ms,0,blend_radius_m)
    |   movel([0.080795, -1.248673, -2.655667, -0.808049, 1.570796, 1.651591],accel_mss,speed_ms,0,blend_radius_m)
    |   movel([0.081727, -1.248356, -2.655835, -0.808198, 1.570796, 1.652524],accel_mss,speed_ms,0,blend_radius_m)
    |   movel([0.082276, -1.248201, -2.655917, -0.808271, 1.570796, 1.653072],accel_mss,speed_ms,0,blend_radius_m)
    |   movel([0.082396, -1.248402, -2.655810, -0.808176, 1.570796, 1.653193],accel_mss,speed_ms,0,blend_radius_m)
    |   movel([0.081838, -1.249465, -2.655246, -0.807678, 1.570796, 1.652635],accel_mss,speed_ms,0,blend_radius_m)
    |   movel([0.081159, -1.250720, -2.654578, -0.807090, 1.570796, 1.651955],accel_mss,speed_ms,0,blend_radius_m)
    |   movel([0.080328, -1.252201, -2.653788, -0.806400, 1.570796, 1.651124],accel_mss,speed_ms,0,blend_radius_m)
    |   movel([0.079241, -1.254128, -2.652755, -0.805506, 1.570796, 1.650037],accel_mss,speed_ms,0,blend_radius_m)
    |   movel([0.078655, -1.255224, -2.652166, -0.804999, 1.570796, 1.649451],accel_mss,speed_ms,0,blend_radius_m)
    |   movel([0.078314, -1.255922, -2.651790, -0.804677, 1.570796, 1.649110],accel_mss,speed_ms,0,blend_radius_m)
    |   movel([0.078472, -1.256172, -2.651655, -0.804562, 1.570796, 1.649269],accel_mss,speed_ms,0,blend_radius_m)
    |   movel([0.078805, -1.256112, -2.651688, -0.804589, 1.570796, 1.649601],accel_mss,speed_ms,0,blend_radius_m)
    |   movel([0.079378, -1.255941, -2.651780, -0.804668, 1.570796, 1.650175],accel_mss,speed_ms,0,blend_radius_m)
    |   movel([0.080470, -1.255566, -2.651982, -0.804841, 1.570796, 1.651266],accel_mss,speed_ms,0,blend_radius_m)
    |   movel([0.081795, -1.255108, -2.652228, -0.805053, 1.570796, 1.652591],accel_mss,speed_ms,0,blend_radius_m)
    |   movel([0.082424, -1.254918, -2.652331, -0.805140, 1.570796, 1.653221],accel_mss,speed_ms,0,blend_radius_m)
    |   movel([0.082757, -1.254859, -2.652362, -0.805167, 1.570796, 1.653553],accel_mss,speed_ms,0,blend_radius_m)
    |   speed_ms = 0.003
    |   movel([0.082807, -1.240828, -2.645414, -0.826147, 1.570796, 1.653603],accel_mss,speed_ms,0,blend_radius_m)
    |   speed_ms = 1.000
    |   movel([0.082807, -1.213918, -2.631313, -0.867159, 1.570796, 1.653603],accel_mss,speed_ms,0,blend_radius_m)
    |   movel([0.061043, -1.170670, -2.652297, -0.889422, 1.570796, 1.631840],accel_mss,speed_ms,0,blend_radius_m)
    |   movel([0.061043, -1.077942, -2.586592, -1.047856, 1.570796, 1.631840],accel_mss,speed_ms,0,blend_radius_m)
    |   # End of main program
    | end
    | 
    | Machining1()
